	(*FB_Gripper Manual*)
		fbGripperManu( // Call Griper mouvement
				eGripperMode:=eGripperMode,
				tMouvementDuration:=tGripperTime,
				bSensorCheck:=bGripperSensor
				);
		IF fbGripperManu.bDone THEN // Gripper Done
			fbGripperManu.bStart:=FALSE;
			(*Log*)
				PRG_Log_WM.fbLogWM.M_Write_Log('MANUAL : Gripper -> DONE');
		ELSIF fbGripperManu.bError THEN // Gripper Error
			//bError:=TRUE;
			//udiErrorID:=?00+fbGripper.udiErrorID; // ?xx = ? + Error xx fbGripperManu
			fbGripperManu.bStart:=FALSE;
			(*Log*)
				PRG_Log_WM.fbLogWM.M_Write_Log('MANUAL : GripperUnclamp -> ERROR');
				PRG_Log_WM.fbLogWM.M_Write_Log(CONCAT('MANUAL : GripperUnclamp : ErrorID=',UDINT_TO_STRING(fbGripperManu.udiErrorID)));
		END_IF
			
(** CHANGING ARM **)
	(*Axis Position*)
		GV_Tool_Magazine.stArm.lrArmPosition:=LINT_TO_LREAL(LREAL_TO_LINT(GV_Axes.stAxisArm.stDriveAx8206.AxisRef.NcToPlc.ActPos*1000.0))/1000.0;
	(*Memory*)
		(*Gripper1*)
			IF GV_Tool_Magazine.stArm.aGripper[1].iAbsLocationNumberMemory<>0 AND GV_Tool_Magazine.stArm.aGripper[1].iRelLocationNumberMemory<>0 THEN
				GV_Tool_Magazine.stArm.aGripper[1].bToolPresenceMemory:=TRUE;
			ELSE
				GV_Tool_Magazine.stArm.aGripper[1].bToolPresenceMemory:=FALSE;
			END_IF
		(*Gripper2*)
			IF GV_Tool_Magazine.stArm.aGripper[2].iAbsLocationNumberMemory<>0 AND GV_Tool_Magazine.stArm.aGripper[2].iRelLocationNumberMemory<>0 THEN
				GV_Tool_Magazine.stArm.aGripper[2].bToolPresenceMemory:=TRUE;
			ELSE
				GV_Tool_Magazine.stArm.aGripper[2].bToolPresenceMemory:=FALSE;
			END_IF
	(*Positions*)
		IF GV_Tool_Magazine.stArm.lrArmPosition<=(GV_Tool_Magazine.stArm.lrArmHome+GV_Tool_Magazine.stArm.lrArmPositionTol) AND GV_Tool_Magazine.stArm.lrArmPosition>=(GV_Tool_Magazine.stArm.lrArmHome-GV_Tool_Magazine.stArm.lrArmPositionTol) THEN
			GV_Tool_Magazine.stArm.ePositionAxis:=ENUM_Position_Axis.Home;
		ELSIF GV_Tool_Magazine.stArm.lrArmPosition<=(GV_Tool_Magazine.stArm.lrArmManipulator+GV_Tool_Magazine.stArm.lrArmPositionTol) AND GV_Tool_Magazine.stArm.lrArmPosition>=(GV_Tool_Magazine.stArm.lrArmManipulator-GV_Tool_Magazine.stArm.lrArmPositionTol) THEN 
			GV_Tool_Magazine.stArm.ePositionAxis:=ENUM_Position_Axis.Work1;
		ELSIF GV_Tool_Magazine.stArm.lrArmPosition<=(GV_Tool_Magazine.stArm.lrArmCNC+GV_Tool_Magazine.stArm.lrArmPositionTol) AND GV_Tool_Magazine.stArm.lrArmPosition>=(GV_Tool_Magazine.stArm.lrArmCNC-GV_Tool_Magazine.stArm.lrArmPositionTol) THEN 
			GV_Tool_Magazine.stArm.ePositionAxis:=ENUM_Position_Axis.CNC;
		ELSE
			GV_Tool_Magazine.stArm.ePositionAxis:=ENUM_Position_Axis.Unknow;
		END_IF

	(*Evacuate*)
		//IF GV_CNC.stFanucData.stCncMagazine.biEvacuateArm AND  THEN
			
		//END_IF

(** TEACHING **)
	(* Selected Location *)
		IF GV_HMI.stMagazineTeach.iTeachLocationSelected>0 AND (GV_HMI.stMagazineTeach.iTeachLocationSelected+1)<=GV_Tool_Magazine.iMaxAbsLocation THEN
			GV_HMI.stMagazineTeach.sTeachLocationSelected:=INT_TO_STRING(GV_Tool_Magazine.aLocation[(GV_HMI.stMagazineTeach.iTeachLocationSelected+1)].iRelLocationNumber);
		END_IF
	
	(* Authorization *)
		GV_Tool_Magazine.bAuthorizationTeachLocation:=(NOT GV_Cycle.bCycleInProgress) AND GV_OpMode.eOpMode=ENUM_OpMode.MANU AND GV_Axes.bAxisAllNotMoving AND (*GV_Axes.bAxisAllOperational AND*) GV_HMI.iCurrentScreenNumber=310 AND GV_HMI.stMagazineTeach.iTeachLocationSelected>0 AND (GV_HMI.stMagazineTeach.iTeachLocationSelected+1)<=GV_Tool_Magazine.iMaxAbsLocation;
		GV_Tool_Magazine.bAuthorizationTeachRack:=(NOT GV_Cycle.bCycleInProgress) AND GV_HMI.iCurrentScreenNumber=310;
		GV_Tool_Magazine.bAuthorizationTeachAllTop:=(NOT GV_Cycle.bCycleInProgress) AND GV_HMI.iCurrentScreenNumber=310;
		GV_Tool_Magazine.bAuthorizationTeachAllBottom:=(NOT GV_Cycle.bCycleInProgress) AND GV_HMI.iCurrentScreenNumber=310;
		GV_Tool_Magazine.bAuthorizationTeachPositions:=(NOT GV_Cycle.bCycleInProgress) AND GV_HMI.iCurrentScreenNumber=311;
	
	(* Limit *)
		IF GV_HMI.stMagazineTeach.iTeachLocationSelected>0 AND (GV_HMI.stMagazineTeach.iTeachLocationSelected+1)<=GV_Tool_Magazine.iMaxAbsLocation THEN
			IF GV_Tool_Magazine.aLocation[(GV_HMI.stMagazineTeach.iTeachLocationSelected+1)].ePositionMag=ENUM_Position_Magazine.Top THEN
				GV_Tool_Magazine.lrMinXTeach:=GV_Tool_Magazine.lrMinXFirstLocationTop;
				GV_Tool_Magazine.lrMaxXTeach:=GV_Tool_Magazine.lrMaxXFirstLocationTop;
				GV_Tool_Magazine.lrMinYTeach:=GV_Tool_Magazine.lrMinYLocationTop;
				GV_Tool_Magazine.lrMaxYTeach:=GV_Tool_Magazine.lrMaxYLocationTop;
				GV_Tool_Magazine.lrMinZTeach:=GV_Tool_Magazine.lrMinZLowestRackTop;
				GV_Tool_Magazine.lrMaxZTeach:=GV_Tool_Magazine.lrMaxZLowestRackTop;
			ELSIF GV_Tool_Magazine.aLocation[(GV_HMI.stMagazineTeach.iTeachLocationSelected+1)].ePositionMag=ENUM_Position_Magazine.Bottom THEN
				GV_Tool_Magazine.lrMinXTeach:=GV_Tool_Magazine.lrMinXFirstLocationBottom;
				GV_Tool_Magazine.lrMaxXTeach:=GV_Tool_Magazine.lrMaxXFirstLocationBottom;
				GV_Tool_Magazine.lrMinYTeach:=GV_Tool_Magazine.lrMinYLocationBottom;
				GV_Tool_Magazine.lrMaxYTeach:=GV_Tool_Magazine.lrMaxYLocationBottom;
				GV_Tool_Magazine.lrMinZTeach:=GV_Tool_Magazine.lrMinZLowestRackBottom;
				GV_Tool_Magazine.lrMaxZTeach:=GV_Tool_Magazine.lrMaxZLowestRackBottom;
			ELSE
				GV_Tool_Magazine.lrMinXTeach:=9999.999;
				GV_Tool_Magazine.lrMaxXTeach:=9999.999;
				GV_Tool_Magazine.lrMinYTeach:=9999.999;
				GV_Tool_Magazine.lrMaxYTeach:=9999.999;
				GV_Tool_Magazine.lrMinZTeach:=9999.999;
				GV_Tool_Magazine.lrMaxZTeach:=9999.999;
			END_IF
		END_IF
		
	(* Teach Location *)
		IF GV_HMI.stMagazineTeach.rtTeachLocation.Q AND GV_Tool_Magazine.bAuthorizationTeachLocation AND GV_HMI.stMagazineTeach.iTeachLocationSelected>0 AND (GV_HMI.stMagazineTeach.iTeachLocationSelected+1)<=GV_Tool_Magazine.iMaxAbsLocation THEN
			GV_Tool_Magazine.aLocation[(GV_HMI.stMagazineTeach.iTeachLocationSelected+1)].lrXcoord:=LINT_TO_LREAL(LREAL_TO_LINT(GV_Axes.stAxisX.stDriveAx8206.AxisRef.NcToPlc.ActPos*1000.0))/1000.0; // Round 10e-3
			GV_Tool_Magazine.aLocation[(GV_HMI.stMagazineTeach.iTeachLocationSelected+1)].lrYcoord:=LINT_TO_LREAL(LREAL_TO_LINT(GV_Axes.stAxisY.stDriveAx8206.AxisRef.NcToPlc.ActPos*1000.0))/1000.0; // Round 10e-3
			GV_Tool_Magazine.aLocation[(GV_HMI.stMagazineTeach.iTeachLocationSelected+1)].lrZcoord:=LINT_TO_LREAL(LREAL_TO_LINT(GV_Axes.stAxisZ.stDriveAx8206.AxisRef.NcToPlc.ActPos*1000.0))/1000.0; // Round 10e-3
		END_IF

	(* Teach Rack *)
		IF GV_HMI.stMagazineTeach.iTeachLocationSelected>0 AND (GV_HMI.stMagazineTeach.iTeachLocationSelected+1)<=GV_Tool_Magazine.iMaxAbsLocation THEN
			
			IF GV_Tool_Magazine.aLocation[(GV_HMI.stMagazineTeach.iTeachLocationSelected+1)].iRelLocationNumber>1 THEN
				IF GV_Tool_Magazine.aLocation[(GV_HMI.stMagazineTeach.iTeachLocationSelected)].iRackNumber<GV_Tool_Magazine.aLocation[(GV_HMI.stMagazineTeach.iTeachLocationSelected+1)].iRackNumber THEN
					GV_HMI.stMagazineTeach.bVisuTeachRack:=TRUE;
				ELSE
					IF GV_Tool_Magazine.aLocation[(GV_HMI.stMagazineTeach.iTeachLocationSelected)].iRackNumber=GV_Tool_Magazine.aLocation[(GV_HMI.stMagazineTeach.iTeachLocationSelected+1)].iRackNumber AND GV_Tool_Magazine.aLocation[(GV_HMI.stMagazineTeach.iTeachLocationSelected)].iRelLocationNumber=0 THEN
						GV_HMI.stMagazineTeach.bVisuTeachRack:=TRUE;
					ELSE
						GV_HMI.stMagazineTeach.bVisuTeachRack:=FALSE;
					END_IF
				END_IF
			ELSE
				IF GV_Tool_Magazine.aLocation[(GV_HMI.stMagazineTeach.iTeachLocationSelected+1)].iRelLocationNumber=1 THEN
					GV_HMI.stMagazineTeach.bVisuTeachRack:=TRUE;
				ELSE
					GV_HMI.stMagazineTeach.bVisuTeachRack:=FALSE;
				END_IF
			END_IF
			
			IF GV_HMI.stMagazineTeach.rtTeachRack.Q AND GV_HMI.stMagazineTeach.bVisuTeachRack AND GV_Tool_Magazine.bAuthorizationTeachRack THEN
				IF GV_Tool_Magazine.aLocation[(GV_HMI.stMagazineTeach.iTeachLocationSelected+1)].ePositionMag=ENUM_Position_magazine.Top THEN
					iCount:=0;
					lrTeachRackZ:=0;
					FOR iTeachLoop:=(GV_HMI.stMagazineTeach.iTeachLocationSelected+1) TO GV_Tool_Magazine.iMaxAbsLocation BY 1 DO
						IF iTeachLoop=(GV_HMI.stMagazineTeach.iTeachLocationSelected+1) THEN
							lrTeachRackZ:=GV_Tool_Magazine.aLocation[(GV_HMI.stMagazineTeach.iTeachLocationSelected+1)].lrZcoord;
						END_IF
						IF GV_Tool_Magazine.aLocation[iTeachLoop].iRackNumber=GV_Tool_Magazine.aLocation[(GV_HMI.stMagazineTeach.iTeachLocationSelected+1)].iRackNumber THEN
							GV_Tool_Magazine.aLocation[iTeachLoop].lrXcoord:=GV_Tool_Magazine.aLocation[(GV_HMI.stMagazineTeach.iTeachLocationSelected+1)].lrXcoord+(GV_Tool_Magazine.lrXLocationOffsetTop*(iTeachLoop-(GV_HMI.stMagazineTeach.iTeachLocationSelected+1)));
								GV_Tool_Magazine.aLocation[iTeachLoop].lrXcoord:=LINT_TO_LREAL(LREAL_TO_LINT(GV_Tool_Magazine.aLocation[iTeachLoop].lrXcoord*1000.0))/1000.0; // Round 10e-3
							GV_Tool_Magazine.aLocation[iTeachLoop].lrYcoord:=GV_Tool_Magazine.aLocation[(GV_HMI.stMagazineTeach.iTeachLocationSelected+1)].lrYcoord+(GV_Tool_Magazine.lrYLocationOffsetTop*(iTeachLoop-(GV_HMI.stMagazineTeach.iTeachLocationSelected+1)));;
								GV_Tool_Magazine.aLocation[iTeachLoop].lrYcoord:=LINT_TO_LREAL(LREAL_TO_LINT(GV_Tool_Magazine.aLocation[iTeachLoop].lrYcoord*1000.0))/1000.0; // Round 10e-3
 							GV_Tool_Magazine.aLocation[iTeachLoop].lrZcoord:=lrTeachRackZ-(GV_Tool_Magazine.lrZRelCompensationLocationTop*iCount); // Compensation
								GV_Tool_Magazine.aLocation[iTeachLoop].lrZcoord:=LINT_TO_LREAL(LREAL_TO_LINT(GV_Tool_Magazine.aLocation[iTeachLoop].lrZcoord*1000.0))/1000.0; // Round 10e-3
							iCount:=iCount+1;
						ELSE
							EXIT;
						END_IF
					END_FOR
				ELSIF GV_Tool_Magazine.aLocation[(GV_HMI.stMagazineTeach.iTeachLocationSelected+1)].ePositionMag=ENUM_Position_magazine.Bottom THEN
					iCount:=0;
					lrTeachRackZ:=0;
					FOR iTeachLoop:=(GV_HMI.stMagazineTeach.iTeachLocationSelected+1) TO GV_Tool_Magazine.iMaxAbsLocation BY 1 DO
						IF iTeachLoop=(GV_HMI.stMagazineTeach.iTeachLocationSelected+1) THEN
							lrTeachRackZ:=GV_Tool_Magazine.aLocation[(GV_HMI.stMagazineTeach.iTeachLocationSelected+1)].lrZcoord;
						END_IF
						IF GV_Tool_Magazine.aLocation[iTeachLoop].iRackNumber=GV_Tool_Magazine.aLocation[(GV_HMI.stMagazineTeach.iTeachLocationSelected+1)].iRackNumber THEN
							GV_Tool_Magazine.aLocation[iTeachLoop].lrXcoord:=GV_Tool_Magazine.aLocation[(GV_HMI.stMagazineTeach.iTeachLocationSelected+1)].lrXcoord+(GV_Tool_Magazine.lrXLocationOffsetBottom*(iTeachLoop-(GV_HMI.stMagazineTeach.iTeachLocationSelected+1)));
								GV_Tool_Magazine.aLocation[iTeachLoop].lrXcoord:=LINT_TO_LREAL(LREAL_TO_LINT(GV_Tool_Magazine.aLocation[iTeachLoop].lrXcoord*1000.0))/1000.0; // Round 10e-3
							GV_Tool_Magazine.aLocation[iTeachLoop].lrYcoord:=GV_Tool_Magazine.aLocation[(GV_HMI.stMagazineTeach.iTeachLocationSelected+1)].lrYcoord+(GV_Tool_Magazine.lrYLocationOffsetBottom*(iTeachLoop-(GV_HMI.stMagazineTeach.iTeachLocationSelected+1)));
								GV_Tool_Magazine.aLocation[iTeachLoop].lrYcoord:=LINT_TO_LREAL(LREAL_TO_LINT(GV_Tool_Magazine.aLocation[iTeachLoop].lrYcoord*1000.0))/1000.0; // Round 10e-3
							GV_Tool_Magazine.aLocation[iTeachLoop].lrZcoord:=lrTeachRackZ-(GV_Tool_Magazine.lrZRelCompensationLocationBottom*iCount); // Compensation
								GV_Tool_Magazine.aLocation[iTeachLoop].lrZcoord:=LINT_TO_LREAL(LREAL_TO_LINT(GV_Tool_Magazine.aLocation[iTeachLoop].lrZcoord*1000.0))/1000.0; // Round 10e-3
							iCount:=iCount+1;
						ELSE
							EXIT;
						END_IF
					END_FOR
				//ELSE
					// Normally not possible to be here -> Can't select from HMI a Location with (ENUM_Position_magazine<>Top OR ENUM_Position_magazine<>Bottom)
				END_IF
			END_IF
			
		END_IF
	
	(* Teach All Top *)
// 		IF GV_HMI.stMagazineTeach.iTeachLocationSelected>0 AND (GV_HMI.stMagazineTeach.iTeachLocationSelected+1)<=GV_Tool_Magazine.iMaxAbsLocation THEN
// 			
// 			IF GV_Tool_Magazine.aLocation[(GV_HMI.stMagazineTeach.iTeachLocationSelected+1)].iRelLocationNumber=1 AND GV_Tool_Magazine.aLocation[(GV_HMI.stMagazineTeach.iTeachLocationSelected+1)].ePositionMag=ENUM_Position_magazine.Top THEN
// 				IF GV_Tool_Magazine.aLocation[(GV_HMI.stMagazineTeach.iTeachLocationSelected+1)].iRackNumber = 1eR Rack du haut THEN
// 					GV_HMI.stMagazineTeach.bVisuTeachAllTop:=TRUE;
// 				ELSE
// 					GV_HMI.stMagazineTeach.bVisuTeachAllTop:=FALSE;
// 				END_IF
// 			ELSE
// 				GV_HMI.stMagazineTeach.bVisuTeachAllTop:=FALSE;
// 			END_IF
// 	
// 			IF GV_HMI.stMagazineTeach.rtTeachAllTop.Q AND GV_HMI.stMagazineTeach.bVisuTeachAllTop AND GV_Tool_Magazine.bAuthorizationTeachAllTop THEN
// 				iCount:=0;
// 				lrTeachAllX:=0.0;
// 				lrTeachAllY:=0.0;
// 				lrTeachAllZ:=0.0;
// 				
// 				
// 				FOR iTeachLoop:=1 TO GV_Tool_Magazine.iMaxAbsLocationTop BY 1 DO
// 					
// 					// Ne pas modifier la position rel 1 car apprise, on part justement de ces valeurs pour recalculer le reste
// 					
// // 					IF iTeachLoop=(GV_HMI.stMagazineTeach.iTeachLocationSelected+1) THEN
// // 						lrTeachRackZ:=GV_Tool_Magazine.aLocation[(GV_HMI.stMagazineTeach.iTeachLocationSelected+1)].lrZcoord;
// // 					END_IF
// // 					IF GV_Tool_Magazine.aLocation[iTeachLoop].iRackNumber=GV_Tool_Magazine.aLocation[(GV_HMI.stMagazineTeach.iTeachLocationSelected+1)].iRackNumber THEN
// // 						GV_Tool_Magazine.aLocation[iTeachLoop].lrXcoord:=GV_Tool_Magazine.aLocation[(GV_HMI.stMagazineTeach.iTeachLocationSelected+1)].lrXcoord+(GV_Tool_Magazine.lrXLocationOffsetTop*(iTeachLoop-(GV_HMI.stMagazineTeach.iTeachLocationSelected+1)));
// // 							GV_Tool_Magazine.aLocation[iTeachLoop].lrXcoord:=LINT_TO_LREAL(LREAL_TO_LINT(GV_Tool_Magazine.aLocation[iTeachLoop].lrXcoord*1000.0))/1000.0; // Round 10e-3
// // 						GV_Tool_Magazine.aLocation[iTeachLoop].lrYcoord:=GV_Tool_Magazine.aLocation[(GV_HMI.stMagazineTeach.iTeachLocationSelected+1)].lrYcoord+(GV_Tool_Magazine.lrYLocationOffsetTop*(iTeachLoop-(GV_HMI.stMagazineTeach.iTeachLocationSelected+1)));;
// // 							GV_Tool_Magazine.aLocation[iTeachLoop].lrYcoord:=LINT_TO_LREAL(LREAL_TO_LINT(GV_Tool_Magazine.aLocation[iTeachLoop].lrYcoord*1000.0))/1000.0; // Round 10e-3
// //  						GV_Tool_Magazine.aLocation[iTeachLoop].lrZcoord:=lrTeachRackZ-(GV_Tool_Magazine.lrZRelCompensationLocationTop*iCount); // Compensation
// // 							GV_Tool_Magazine.aLocation[iTeachLoop].lrZcoord:=LINT_TO_LREAL(LREAL_TO_LINT(GV_Tool_Magazine.aLocation[iTeachLoop].lrZcoord*1000.0))/1000.0; // Round 10e-3
// // 						iCount:=iCount+1;
// // 					ELSE
// // 						EXIT;
// // 					END_IF
// 				END_FOR
// 				
// 				
// 				
// 			END_IF
// 	
// 		END_IF

	(* Teach All Bottom *)

END_PROGRAM

// ---- 09_Tool_Magazine/03_POUs/02_FBs/FB_Manipulator_Tunnel_5.TcPOU
FUNCTION_BLOCK FB_Manipulator_Tunnel_5
VAR_INPUT
	(** SETUP ENUM **)
		eTunnelMode : ENUM_Tunnel_Mode ; // Mode of the tunnel	

	(** SETUP TIME **)
		tTimeout : TIME ; // Max time for travel the tunnel

	(** PROCESS FLAG **)
		bInit : BOOL ; // Init the FB
	    bStart : BOOL ; // Start the Fb
END_VAR
VAR_OUTPUT
	(** PROCESS UDINT **)
		udiErrorID : UDINT ; // Fb Error ID
		
	(** PROCESS FLAG **)
		bBusy  : BOOL ; // Fb is Busy
		bDone  : BOOL ; // Fb is Done
		bError : BOOL ; // Fb in Error
END_VAR
VAR_IN_OUT
END_VAR	
VAR
	(** STRING **)
		strTextLog : STRING ; // Text to Log

	(** PROCESS INT **)
		iStep  : INT := 0 ; // Step of the Fb
		iSubStep : INT := 0 ; // SubStep of the Fb
		iPrevStep : INT := 0 ; // Previous Step of the Fb
		iPrevSubStep : INT := 0 ; // Previous Subtep of the Fb
	
	(** PROCESS FLAG + R_TRIG **)
		rtInit : R_TRIG ; // FB Init at rising edge
		rtStart : R_TRIG ; // FB Start at rising edge
		bTunnelTravelDone : BOOL ; // Tunnel travel done
		bXError : BOOL ; // Axis X Error
		bYError : BOOL ; // Axis Y Error
		bZError : BOOL ; // Axis Z Error
		bArmError : BOOL ; // Axis Arm Error
		
	(** FB **)
		tonTimeout : TON ; // TON timeout of the tunnel travel
END_VAR

//-----------------------------------------------------------------------------------------
//
//                  		FB_Manipulator_Tunnel
//
//			Management of the manipulator passage through the tunnel
//-----------------------------------------------------------------------------------------
//
//Auteur: G.GOETZ
//Création: 06.02.2026
//Dernière modification : 08.04.2026 (G.GOETZ)
//       			
//-----------------------------------------------------------------------------------------
//
//     							Liste des modifications  	
//
// 06.02.2026 (G.GOETZ) -> Création
// 08.04.2026 (G.GOETZ) -> Ajout Init + Modification du cycle
//-----------------------------------------------------------------------------------------

(** FB CALL **)
	rtInit(CLK:=bInit);
	rtStart(CLK:=bStart);
	
	tonTimeout();

(** AXIS ERRORS **)
	bXError:=(GV_Axes.stAxisX.stDriveAx8206.AxisRef.Status.Error OR GV_Axes.stAxisX.stDriveAx8206.AxisRef.Status.ErrorStop OR GV_Axes.stAxisX.stDriveAx8206.AxisRef.Status.ErrorID<>0);
	bYError:=(GV_Axes.stAxisY.stDriveAx8206.AxisRef.Status.Error OR GV_Axes.stAxisY.stDriveAx8206.AxisRef.Status.ErrorStop OR GV_Axes.stAxisY.stDriveAx8206.AxisRef.Status.ErrorID<>0);
	bZError:=(GV_Axes.stAxisZ.stDriveAx8206.AxisRef.Status.Error OR GV_Axes.stAxisZ.stDriveAx8206.AxisRef.Status.ErrorStop OR GV_Axes.stAxisZ.stDriveAx8206.AxisRef.Status.ErrorID<>0);
	bArmError:=(GV_Axes.stAxisArm.stDriveAx8206.AxisRef.Status.Error OR GV_Axes.stAxisArm.stDriveAx8206.AxisRef.Status.ErrorStop OR GV_Axes.stAxisArm.stDriveAx8206.AxisRef.Status.ErrorID<>0);

(** INIT **)
	IF (rtinit.Q OR bInit) AND (NOT bStart) THEN
		iStep:=0;
		bInit:=FALSE;
	END_IF

(** STEPS **)
    CASE iStep OF
		
        0: (* Step 0 = Idle *)
            bBusy:=FALSE;
            bDone:=FALSE;
			bError:=FALSE;
			udiErrorID:=0;
			iSubStep:=0;
			
			tonTimeout.IN:=FALSE;
			
			bTunnelTravelDone:=FALSE;
			
			(* Idle->Setup *)
				IF bStart AND (NOT bInit) THEN
					bBusy:=TRUE;
					(*Log*)
						PRG_Log_WM.fbLogWM.M_Write_Log('FB_Manipulator_Tunnel : 0_Idle->1_Setup');
					iStep:=1; // Next Step
				END_IF
				
		1: (* Step 1 = Setup *)
			(*Log*)
				(*TunnelMode*)
					CASE eTunnelMode OF
						ENUM_Tunnel_Mode.TopToBottom:		strTextLog:='TopToBottom';
						ENUM_Tunnel_Mode.BottomToTop:		strTextLog:='BottomToTop';
					END_CASE
					PRG_Log_WM.fbLogWM.M_Write_Log(CONCAT('FB_Manipulator_Tunnel : 1_Setup : Tunnel Mode = ',strTextLog));
				(*Timeout*)
					strTextLog:=TIME_TO_STRING(tTimeout);
					PRG_Log_WM.fbLogWM.M_Write_Log(CONCAT('FB_Manipulator_Tunnel : 1_Setup : Timeout = ',strTextLog));				
				PRG_Log_WM.fbLogWM.M_Write_Log('FB_Manipulator_Tunnel : 1_Setup->2_Process');
				
			tonTimeout.PT:=tTimeout;
			iStep:=2; // Next Step
			
		2: (* Step 2 = Process (Y->(XFirst)->Z->X) *) // -> (* Step 2 = Process (Y->(ZLowestRacKTop)->(XFirst)) *) + (* Step 3 = Process (Z->X) *)	
			tonTimeout.IN:=TRUE; // Start TON timeout

				CASE iSubStep OF
		
					0: (* Start Y move *)
						GV_Axes.stAxisY.lrAutoPosAbs:=GV_Tool_Magazine.stManipulator.lrYTunnel;
						GV_Axes.stAxisY.bAutoCmdAbs:=TRUE;
						(*Log*)
							PRG_Log_WM.fbLogWM.M_Write_Log('FB_Manipulator_Tunnel : 2_Process : 0 : Start Y move');
						iSubStep:=1; // Next SubStep
						
					1: (* Wait Y move done *)
					   IF GV_Axes.stAxisY.bAutoDone AND (NOT bYError) THEN
							GV_Axes.stAxisY.bAutoCmdAbs:=FALSE;
							(*Log*)
								PRG_Log_WM.fbLogWM.M_Write_Log('FB_Manipulator_Tunnel : 2_Process : 1 : Y move done');

							CASE eTunnelMode OF 
								ENUM_Tunnel_Mode.TopToBottom: // X Top
									IF GV_Tool_Magazine.stManipulator.lrXPosition<GV_Tool_Magazine.lrXFirstLocationTop THEN
										(*Log*)
											PRG_Log_WM.fbLogWM.M_Write_Log('FB_Manipulator_Tunnel : 2_Process : 1->2 : XFirstTop');
										iSubStep:=2; // Next SubStep
									ELSE
										(*Log*)
											PRG_Log_WM.fbLogWM.M_Write_Log('FB_Manipulator_Tunnel : 2_Process : 1->4 : Z');
										iSubStep:=4; // Next SubStep
									END_IF
								ENUM_Tunnel_Mode.BottomToTop: // X Bottom
									IF GV_Tool_Magazine.stManipulator.lrXPosition<GV_Tool_Magazine.lrXFirstLocationBottom THEN
										(*Log*)
											PRG_Log_WM.fbLogWM.M_Write_Log('FB_Manipulator_Tunnel : 2_Process : 1->2 : XFirstBottom');
										iSubStep:=2; // Next SubStep
									ELSE
										(*Log*)
											PRG_Log_WM.fbLogWM.M_Write_Log('FB_Manipulator_Tunnel : 2_Process : 1->4 : Z');
										iSubStep:=4; // Next SubStep
									END_IF
							END_CASE
						ELSIF bYError THEN
							bError:=TRUE;
							udiErrorID:=21; // 21 = Step 2 SubStep 1 Error Axis Y
							GV_Axes.stAxisY.bAutoCmdAbs:=FALSE;
							tonTimeout.IN:=FALSE;
							(*Log*)
								PRG_Log_WM.fbLogWM.M_Write_Log('FB_Manipulator_Tunnel : 2_Process=Error');
								PRG_Log_WM.fbLogWM.M_Write_Log(CONCAT('FB_Manipulator_Tunnel : ErrorID=',UDINT_TO_STRING(udiErrorID)));
							iSubStep:=0; // Stop SubStep
							iStep:=0; // Idle Step
						END_IF
						
					2: (* Start XFirst move *)
						CASE eTunnelMode OF 
							ENUM_Tunnel_Mode.TopToBottom: // X Top
								GV_Axes.stAxisX.lrAutoPosAbs:=GV_Tool_Magazine.lrXFirstLocationTop;
								(*Log*)
									PRG_Log_WM.fbLogWM.M_Write_Log('FB_Manipulator_Tunnel : 2_Process : 2 : Start XFirstTop move');
							ENUM_Tunnel_Mode.BottomToTop: // X Bottom
								GV_Axes.stAxisX.lrAutoPosAbs:=GV_Tool_Magazine.lrXFirstLocationBottom;
								(*Log*)
									PRG_Log_WM.fbLogWM.M_Write_Log('FB_Manipulator_Tunnel : 2_Process : 2 : Start XFirstBottom move');
						END_CASE
						GV_Axes.stAxisX.bAutoCmdAbs:=TRUE;
						iSubStep:=3; // Next SubStep

					3: (* Wait XFirst move done *)
					   IF GV_Axes.stAxisX.bAutoDone AND (NOT bXError) THEN
							GV_Axes.stAxisX.bAutoCmdAbs:=FALSE;
							(*Log*)
								PRG_Log_WM.fbLogWM.M_Write_Log('FB_Manipulator_Tunnel : 2_Process : 3 : XFirst move done');
							iSubStep:=4; // Next SubStep
						ELSIF bXError THEN
							bError:=TRUE;
							udiErrorID:=23; // 23 = Step 2 SubStep 3 Error Axis X
							GV_Axes.stAxisX.bAutoCmdAbs:=FALSE;
							tonTimeout.IN:=FALSE;
							(*Log*)
								PRG_Log_WM.fbLogWM.M_Write_Log('FB_Manipulator_Tunnel : 2_Process=Error');
								PRG_Log_WM.fbLogWM.M_Write_Log(CONCAT('FB_Manipulator_Tunnel : ErrorID=',UDINT_TO_STRING(udiErrorID)));
							iSubStep:=0; // Stop 
							iStep:=0; // Idle Step
						END_IF
						
					4: (* Start Z move *)
						CASE eTunnelMode OF 
							ENUM_Tunnel_Mode.TopToBottom: // Z bottom position
								GV_Axes.stAxisZ.lrAutoPosAbs:=GV_Tool_Magazine.stManipulator.lrZTunnelBottom;
							ENUM_Tunnel_Mode.BottomToTop: // Z top position
								GV_Axes.stAxisZ.lrAutoPosAbs:=GV_Tool_Magazine.stManipulator.lrZTunnelTop;
						END_CASE
						IF (GV_Axes.stAxisZ.lrAutoPosAbs=GV_Tool_Magazine.stManipulator.lrZTunnelBottom) OR (GV_Axes.stAxisZ.lrAutoPosAbs=GV_Tool_Magazine.stManipulator.lrZTunnelTop) THEN
							GV_Axes.stAxisZ.bAutoCmdAbs:=TRUE;
						ELSE
							GV_Axes.stAxisZ.bAutoCmdAbs:=FALSE;
						END_IF
						(*Log*)
							PRG_Log_WM.fbLogWM.M_Write_Log('FB_Manipulator_Tunnel : 2_Process : 4 : Start Z move');
						iSubStep:=5; // Next Step
		
					5: (* Wait Z move done *)
					   IF GV_Axes.stAxisZ.bAutoDone AND (NOT bZError) THEN
							GV_Axes.stAxisZ.bAutoCmdAbs:=FALSE;
							tonTimeout.IN:=FALSE;
							(*Log*)
								PRG_Log_WM.fbLogWM.M_Write_Log('FB_Manipulator_Tunnel : 2_Process : 5 : Z move done');
							iSubStep:=6; // End SubStep
						ELSIF bZError THEN
							bError:=TRUE;
							udiErrorID:=25; // 25 = Step 2 SubStep 5 Error Axis Z
							GV_Axes.stAxisZ.bAutoCmdAbs:=FALSE;
							tonTimeout.IN:=FALSE;
							(*Log*)
								PRG_Log_WM.fbLogWM.M_Write_Log('FB_Manipulator_Tunnel : 2_Process=Error');
								PRG_Log_WM.fbLogWM.M_Write_Log(CONCAT('FB_Manipulator_Tunnel : ErrorID=',UDINT_TO_STRING(udiErrorID)));
							iSubStep:=0; // Stop SubStep
							iStep:=0; // Idle Step
						END_IF
						
					6: (* Start X move *)
						GV_Axes.stAxisX.lrAutoPosAbs:=GV_Tool_Magazine.stManipulator.lrXTunnel;
						GV_Axes.stAxisX.bAutoCmdAbs:=TRUE;
						(*Log*)
							PRG_Log_WM.fbLogWM.M_Write_Log('FB_Manipulator_Tunnel : 2_Process : 6 : Start X move');
						iSubStep:=7; // Next SubStep
		
					7: (* Wait X move done *)
					   IF GV_Axes.stAxisX.bAutoDone AND (NOT bXError) THEN
							GV_Axes.stAxisX.bAutoCmdAbs:=FALSE;
							(*Log*)
								PRG_Log_WM.fbLogWM.M_Write_Log('FB_Manipulator_Tunnel : 2_Process : 7 : X move done');
							bTunnelTravelDone:=TRUE;
							iSubStep:=0; // Next SubStep
						ELSIF bXError THEN
							bError:=TRUE;
							udiErrorID:=27; // 27 = Step 2 SubStep 7 Error Axis X
							GV_Axes.stAxisX.bAutoCmdAbs:=FALSE;
							tonTimeout.IN:=FALSE;
							(*Log*)
								PRG_Log_WM.fbLogWM.M_Write_Log('FB_Manipulator_Tunnel : 2_Process=Error');
								PRG_Log_WM.fbLogWM.M_Write_Log(CONCAT('FB_Manipulator_Tunnel : ErrorID=',UDINT_TO_STRING(udiErrorID)));
							iSubStep:=0; // Stop SubStep
							iStep:=0; // Idle Step
						END_IF

					END_CASE
			
			IF bTunnelTravelDone THEN
				tonTimeout.IN:=FALSE;
				(*Log*)
					PRG_Log_WM.fbLogWM.M_Write_Log('FB_Manipulator_Tunnel : 2_Process : Done with success');
					PRG_Log_WM.fbLogWM.M_Write_Log('FB_Manipulator_Tunnel : 2_Process->0_Idle');
				iSubStep:=0; // End SubStep
				iStep:=0; // Idle Step
				bDone:=TRUE;
				bBusy:=FALSE;
			END_IF
			
			IF tonTimeout.Q AND tonTimeout.PT<>T#0S THEN
				bError:=TRUE;
				udiErrorID:=29; // 29 = Step 2 Error Timeout 9
				GV_Axes.stAxisZ.bAutoCmdAbs:=FALSE;
				GV_Axes.stAxisX.bAutoCmdAbs:=FALSE;
				GV_Axes.stAxisY.bAutoCmdAbs:=FALSE;
				tonTimeout.IN:=FALSE;
				(*Log*)
					PRG_Log_WM.fbLogWM.M_Write_Log('FB_Manipulator_Tunnel : 2_Process : Error');
					PRG_Log_WM.fbLogWM.M_Write_Log(CONCAT('FB_Manipulator_Tunnel : ErrorID = ',UDINT_TO_STRING(udiErrorID)));
				iSubStep:=0; // Stop SubStep
				iStep:=0; // Idle Step
			END_IF
			
	END_CASE

END_FUNCTION_BLOCK

// ---- 09_Tool_Magazine/03_POUs/02_FBs/FB_Manipulator_Tunnel_2.TcPOU
FUNCTION_BLOCK FB_Manipulator_Tunnel_2
VAR_INPUT
	(** SETUP ENUM **)
		eTunnelMode : ENUM_Tunnel_Mode ; // Mode of the tunnel	

	(** SETUP TIME **)
		tTimeout : TIME ; // Max time for travel the tunnel

	(** PROCESS FLAG **)
		bInit : BOOL ; // Init the FB
	    bStart : BOOL ; // Start the Fb
END_VAR
VAR_OUTPUT
	(** PROCESS UDINT **)
		udiErrorID : UDINT ; // Fb Error ID
		
	(** PROCESS FLAG **)
		bBusy  : BOOL ; // Fb is Busy
		bDone  : BOOL ; // Fb is Done
		bError : BOOL ; // Fb in Error
END_VAR
VAR_IN_OUT
END_VAR	
VAR
	(** STRING **)
		strTextLog : STRING ; // Text to Log

	(** PROCESS INT **)
		iStep  : INT := 0 ; // Step of the Fb
		iSubStep : INT := 0 ; // SubStep of the Fb
		iPrevStep : INT := 0 ; // Previous Step of the Fb
		iPrevSubStep : INT := 0 ; // Previous Subtep of the Fb
	
	(** PROCESS FLAG + R_TRIG **)
		rtInit : R_TRIG ; // FB Init at rising edge
		rtStart : R_TRIG ; // FB Start at rising edge
		bTunnelTravelDone : BOOL ; // Tunnel travel done
		bXError : BOOL ; // Axis X Error
		bYError : BOOL ; // Axis Y Error
		bZError : BOOL ; // Axis Z Error
		bArmError : BOOL ; // Axis Arm Error
		
	(** FB **)
		tonTimeout : TON ; // TON timeout of the tunnel travel
END_VAR

//-----------------------------------------------------------------------------------------
//
//                  		FB_Manipulator_Tunnel
//
//			Management of the manipulator passage through the tunnel
//-----------------------------------------------------------------------------------------
//
//Auteur: G.GOETZ
//Création: 06.02.2026
//Dernière modification : 08.04.2026 (G.GOETZ)
//       			
//-----------------------------------------------------------------------------------------
//
//     							Liste des modifications  	
//
// 06.02.2026 (G.GOETZ) -> Création
// 08.04.2026 (G.GOETZ) -> Ajout Init + Modification du cycle
//-----------------------------------------------------------------------------------------

(** FB CALL **)
	rtInit(CLK:=bInit);
	rtStart(CLK:=bStart);
	
	tonTimeout();

(** AXIS ERRORS **)
	bXError:=(GV_Axes.stAxisX.stDriveAx8206.AxisRef.Status.Error OR GV_Axes.stAxisX.stDriveAx8206.AxisRef.Status.ErrorStop OR GV_Axes.stAxisX.stDriveAx8206.AxisRef.Status.ErrorID<>0);
	bYError:=(GV_Axes.stAxisY.stDriveAx8206.AxisRef.Status.Error OR GV_Axes.stAxisY.stDriveAx8206.AxisRef.Status.ErrorStop OR GV_Axes.stAxisY.stDriveAx8206.AxisRef.Status.ErrorID<>0);
	bZError:=(GV_Axes.stAxisZ.stDriveAx8206.AxisRef.Status.Error OR GV_Axes.stAxisZ.stDriveAx8206.AxisRef.Status.ErrorStop OR GV_Axes.stAxisZ.stDriveAx8206.AxisRef.Status.ErrorID<>0);
	bArmError:=(GV_Axes.stAxisArm.stDriveAx8206.AxisRef.Status.Error OR GV_Axes.stAxisArm.stDriveAx8206.AxisRef.Status.ErrorStop OR GV_Axes.stAxisArm.stDriveAx8206.AxisRef.Status.ErrorID<>0);

(** INIT **)
	IF (rtinit.Q OR bInit) AND (NOT bStart) THEN
		iStep:=0;
		bInit:=FALSE;
	END_IF

(** STEPS **)
    CASE iStep OF
		
        0: (* Step 0 = Idle *)
            bBusy:=FALSE;
            bDone:=FALSE;
			bError:=FALSE;
			udiErrorID:=0;
			iSubStep:=0;
			
			tonTimeout.IN:=FALSE;
			
			bTunnelTravelDone:=FALSE;
			
			(* Idle->Setup *)
				IF bStart AND (NOT bInit) THEN
					bBusy:=TRUE;
					(*Log*)
						PRG_Log_WM.fbLogWM.M_Write_Log('FB_Manipulator_Tunnel : 0_Idle->1_Setup');
					iStep:=1; // Next Step
				END_IF
				
		1: (* Step 1 = Setup *)
			(*Log*)
				(*TunnelMode*)
					CASE eTunnelMode OF
						ENUM_Tunnel_Mode.TopToBottom:		strTextLog:='TopToBottom';
						ENUM_Tunnel_Mode.BottomToTop:		strTextLog:='BottomToTop';
					END_CASE
					PRG_Log_WM.fbLogWM.M_Write_Log(CONCAT('FB_Manipulator_Tunnel : 1_Setup : Tunnel Mode = ',strTextLog));
				(*Timeout*)
					strTextLog:=TIME_TO_STRING(tTimeout);
					PRG_Log_WM.fbLogWM.M_Write_Log(CONCAT('FB_Manipulator_Tunnel : 1_Setup : Timeout = ',strTextLog));				
				PRG_Log_WM.fbLogWM.M_Write_Log('FB_Manipulator_Tunnel : 1_Setup->2_Process');
				
			tonTimeout.PT:=tTimeout;
			iStep:=2; // Next Step
			
		2: (* Step 2 = Process (Y->(ZLowestRacKTop)->(XFirst)) *)
			tonTimeout.IN:=TRUE; // Start TON timeout

				CASE iSubStep OF
		
					0: (* Start Y move *)
						GV_Axes.stAxisY.lrAutoPosAbs:=GV_Tool_Magazine.stManipulator.lrYTunnel;
						GV_Axes.stAxisY.bAutoCmdAbs:=TRUE;
						(*Log*)
							PRG_Log_WM.fbLogWM.M_Write_Log('FB_Manipulator_Tunnel : 2_Process : 0 : Start Y move');
						iSubStep:=1; // Next SubStep
						
					1: (* Wait Y move done *)
					   IF GV_Axes.stAxisY.bAutoDone AND (NOT bYError) THEN
							GV_Axes.stAxisY.bAutoCmdAbs:=FALSE;
							(*Log*)
								PRG_Log_WM.fbLogWM.M_Write_Log('FB_Manipulator_Tunnel : 2_Process : 1 : Y move done');

							CASE eTunnelMode OF 
								ENUM_Tunnel_Mode.TopToBottom: // X Top
									IF GV_Tool_Magazine.stManipulator.lrZPosition<GV_Tool_Magazine.lrZLowestRackTop THEN
										(*Log*)
											PRG_Log_WM.fbLogWM.M_Write_Log('FB_Manipulator_Tunnel : 2_Process : 1->2 : ZLowestRackTop');
										iSubStep:=2; // Next SubStep
									ELSE
										IF GV_Tool_Magazine.stManipulator.lrXPosition<GV_Tool_Magazine.lrXFirstLocationTop THEN
											(*Log*)
												PRG_Log_WM.fbLogWM.M_Write_Log('FB_Manipulator_Tunnel : 2_Process : 1->4 : XFirstTop');
											iSubStep:=4; // Next SubStep
										ELSE
											(*Log*)
												PRG_Log_WM.fbLogWM.M_Write_Log('FB_Manipulator_Tunnel : 2_Process -> 3_Process');
											iSubStep:=0; // End SubStep
											iStep:=3; // Next Stpe
										END_IF
									END_IF
								ENUM_Tunnel_Mode.BottomToTop: // X Bottom
									IF GV_Tool_Magazine.stManipulator.lrXPosition<GV_Tool_Magazine.lrXFirstLocationBottom+GV_Tool_Magazine.lrXLocationOffsetBottom THEN
										(*Log*)
											PRG_Log_WM.fbLogWM.M_Write_Log('FB_Manipulator_Tunnel : 2_Process : 1->4 : XFirstBottom');
										iSubStep:=4; // Next SubStep
									ELSE
										(*Log*)
											PRG_Log_WM.fbLogWM.M_Write_Log('FB_Manipulator_Tunnel : 2_Process -> 3_Process');
											iSubStep:=0; // End SubStep
											iStep:=3; // Next Stpe
									END_IF
							END_CASE
						ELSIF bYError THEN
							bError:=TRUE;
							udiErrorID:=21; // 21 = Step 2 SubStep 1 Error Axis Y
							GV_Axes.stAxisY.bAutoCmdAbs:=FALSE;
							tonTimeout.IN:=FALSE;
							(*Log*)
								PRG_Log_WM.fbLogWM.M_Write_Log('FB_Manipulator_Tunnel : 2_Process=Error');
								PRG_Log_WM.fbLogWM.M_Write_Log(CONCAT('FB_Manipulator_Tunnel : ErrorID=',UDINT_TO_STRING(udiErrorID)));
							iSubStep:=0; // Stop SubStep
							iStep:=0; // Idle Step
						END_IF

					2: (* Start ZLowestRacckTop move *)
						GV_Axes.stAxisZ.lrAutoPosAbs:=GV_Tool_Magazine.lrZLowestRackTop;
						(*Log*)
							PRG_Log_WM.fbLogWM.M_Write_Log('FB_Manipulator_Tunnel : 2_Process : 2 : Start ZLowestRacckTop move');
						GV_Axes.stAxisZ.bAutoCmdAbs:=TRUE;
						iSubStep:=3; // Next SubStep

					3: (* Wait ZLowestRacckTop move done *)
					   IF GV_Axes.stAxisZ.bAutoDone AND (NOT bZError) THEN
							GV_Axes.stAxisZ.bAutoCmdAbs:=FALSE;
							(*Log*)
								PRG_Log_WM.fbLogWM.M_Write_Log('FB_Manipulator_Tunnel : 2_Process : 3 : ZLowestRacckTop move done');
							iSubStep:=0; // End SubStep
							iStep:=4; // Next STep
						ELSIF bZError THEN
							bError:=TRUE;
							udiErrorID:=23; // 23 = Step 2 SubStep 3 Error Axis Z
							GV_Axes.stAxisZ.bAutoCmdAbs:=FALSE;
							tonTimeout.IN:=FALSE;
							(*Log*)
								PRG_Log_WM.fbLogWM.M_Write_Log('FB_Manipulator_Tunnel : 2_Process=Error');
								PRG_Log_WM.fbLogWM.M_Write_Log(CONCAT('FB_Manipulator_Tunnel : ErrorID=',UDINT_TO_STRING(udiErrorID)));
							iSubStep:=0; // Stop 
							iStep:=0; // Idle Step
						END_IF
						
					4: (* Start XFirst move *)
						CASE eTunnelMode OF 
							ENUM_Tunnel_Mode.TopToBottom: // X Top
								GV_Axes.stAxisX.lrAutoPosAbs:=GV_Tool_Magazine.lrXFirstLocationTop;
								(*Log*)
									PRG_Log_WM.fbLogWM.M_Write_Log('FB_Manipulator_Tunnel : 2_Process : 4 : Start XFirstTop move');
							ENUM_Tunnel_Mode.BottomToTop: // X Bottom
								GV_Axes.stAxisX.lrAutoPosAbs:=GV_Tool_Magazine.lrXFirstLocationBottom+GV_Tool_Magazine.lrXLocationOffsetBottom;
								(*Log*)
									PRG_Log_WM.fbLogWM.M_Write_Log('FB_Manipulator_Tunnel : 2_Process : 4 : Start XFirstBottom move');
						END_CASE
						GV_Axes.stAxisX.bAutoCmdAbs:=TRUE;
						iSubStep:=5; // Next SubStep

					5: (* Wait XFirst move done *)
					   IF GV_Axes.stAxisX.bAutoDone AND (NOT bXError) THEN
							GV_Axes.stAxisX.bAutoCmdAbs:=FALSE;
							(*Log*)
								PRG_Log_WM.fbLogWM.M_Write_Log('FB_Manipulator_Tunnel : 2_Process : 5 : XFirst move done');
							iSubStep:=0; // End SubStep
							iStep:=3; // Next STep
						ELSIF bXError THEN
							bError:=TRUE;
							udiErrorID:=25; // 25 = Step 2 SubStep 5 Error Axis X
							GV_Axes.stAxisX.bAutoCmdAbs:=FALSE;
							tonTimeout.IN:=FALSE;
							(*Log*)
								PRG_Log_WM.fbLogWM.M_Write_Log('FB_Manipulator_Tunnel : 2_Process=Error');
								PRG_Log_WM.fbLogWM.M_Write_Log(CONCAT('FB_Manipulator_Tunnel : ErrorID=',UDINT_TO_STRING(udiErrorID)));
							iSubStep:=0; // Stop 
							iStep:=0; // Idle Step
						END_IF
						
				END_CASE
				
			IF tonTimeout.Q AND tonTimeout.PT<>T#0S THEN
				bError:=TRUE;
				udiErrorID:=29; // 29 = Step 2 Error Timeout 9
				GV_Axes.stAxisZ.bAutoCmdAbs:=FALSE;
				GV_Axes.stAxisX.bAutoCmdAbs:=FALSE;
				GV_Axes.stAxisY.bAutoCmdAbs:=FALSE;
				tonTimeout.IN:=FALSE;
				(*Log*)
					PRG_Log_WM.fbLogWM.M_Write_Log('FB_Manipulator_Tunnel : 2_Process : Error');
					PRG_Log_WM.fbLogWM.M_Write_Log(CONCAT('FB_Manipulator_Tunnel : ErrorID = ',UDINT_TO_STRING(udiErrorID)));
				iSubStep:=0; // Stop SubStep
				iStep:=0; // Idle Step
			END_IF
			
		3: (* Step 3 = Process (Z->X) *)	
				CASE iSubStep OF

					0: (* Start Z move *)
						CASE eTunnelMode OF 
							ENUM_Tunnel_Mode.TopToBottom: // Z bottom position
								GV_Axes.stAxisZ.lrAutoPosAbs:=GV_Tool_Magazine.stManipulator.lrZTunnelBottom;
							ENUM_Tunnel_Mode.BottomToTop: // Z top position
								GV_Axes.stAxisZ.lrAutoPosAbs:=GV_Tool_Magazine.stManipulator.lrZTunnelTop;
						END_CASE
						IF (GV_Axes.stAxisZ.lrAutoPosAbs=GV_Tool_Magazine.stManipulator.lrZTunnelBottom) OR (GV_Axes.stAxisZ.lrAutoPosAbs=GV_Tool_Magazine.stManipulator.lrZTunnelTop) THEN
							GV_Axes.stAxisZ.bAutoCmdAbs:=TRUE;
						ELSE
							GV_Axes.stAxisZ.bAutoCmdAbs:=FALSE;
						END_IF
						(*Log*)
							PRG_Log_WM.fbLogWM.M_Write_Log('FB_Manipulator_Tunnel : 3_Process : 0 : Start Z move');
						iSubStep:=1; // Next Step
		
					1: (* Wait Z move done *)
					   IF GV_Axes.stAxisZ.bAutoDone AND (NOT bZError) THEN
							GV_Axes.stAxisZ.bAutoCmdAbs:=FALSE;
							tonTimeout.IN:=FALSE;
							(*Log*)
								PRG_Log_WM.fbLogWM.M_Write_Log('FB_Manipulator_Tunnel : 2_Process : 1 : Z move done');
							iSubStep:=2; // End SubStep
						ELSIF bZError THEN
							bError:=TRUE;
							udiErrorID:=31; // 31 = Step 3 SubStep 1 Error Axis Z
							GV_Axes.stAxisZ.bAutoCmdAbs:=FALSE;
							tonTimeout.IN:=FALSE;
							(*Log*)
								PRG_Log_WM.fbLogWM.M_Write_Log('FB_Manipulator_Tunnel : 3_Process=Error');
								PRG_Log_WM.fbLogWM.M_Write_Log(CONCAT('FB_Manipulator_Tunnel : ErrorID=',UDINT_TO_STRING(udiErrorID)));
							iSubStep:=0; // Stop SubStep
							iStep:=0; // Idle Step
						END_IF
						
					2: (* Start X move *)
						GV_Axes.stAxisX.lrAutoPosAbs:=GV_Tool_Magazine.stManipulator.lrXTunnel;
						GV_Axes.stAxisX.bAutoCmdAbs:=TRUE;
						(*Log*)
							PRG_Log_WM.fbLogWM.M_Write_Log('FB_Manipulator_Tunnel : 3_Process : 2 : Start X move');
						iSubStep:=7; // Next SubStep
		
					3: (* Wait X move done *)
					   IF GV_Axes.stAxisX.bAutoDone AND (NOT bXError) THEN
							GV_Axes.stAxisX.bAutoCmdAbs:=FALSE;
							(*Log*)
								PRG_Log_WM.fbLogWM.M_Write_Log('FB_Manipulator_Tunnel : 3_Process : 3 : X move done');
							bTunnelTravelDone:=TRUE;
							iSubStep:=0; // Next SubStep
						ELSIF bXError THEN
							bError:=TRUE;
							udiErrorID:=33; // 33 = Step 3 SubStep 3 Error Axis X
							GV_Axes.stAxisX.bAutoCmdAbs:=FALSE;
							tonTimeout.IN:=FALSE;
							(*Log*)
								PRG_Log_WM.fbLogWM.M_Write_Log('FB_Manipulator_Tunnel : 3_Process=Error');
								PRG_Log_WM.fbLogWM.M_Write_Log(CONCAT('FB_Manipulator_Tunnel : ErrorID=',UDINT_TO_STRING(udiErrorID)));
							iSubStep:=0; // Stop SubStep
							iStep:=0; // Idle Step
						END_IF

					END_CASE
			
			IF bTunnelTravelDone THEN
				tonTimeout.IN:=FALSE;
				(*Log*)
					PRG_Log_WM.fbLogWM.M_Write_Log('FB_Manipulator_Tunnel : 2_Process : Done with success');
					PRG_Log_WM.fbLogWM.M_Write_Log('FB_Manipulator_Tunnel : 2_Process->0_Idle');
				iSubStep:=0; // End SubStep
				iStep:=0; // Idle Step
				bDone:=TRUE;
				bBusy:=FALSE;
			END_IF
			
			IF tonTimeout.Q AND tonTimeout.PT<>T#0S THEN
				bError:=TRUE;
				udiErrorID:=39; // 39 = Step 3 Error Timeout 9
				GV_Axes.stAxisZ.bAutoCmdAbs:=FALSE;
				GV_Axes.stAxisX.bAutoCmdAbs:=FALSE;
				GV_Axes.stAxisY.bAutoCmdAbs:=FALSE;
				tonTimeout.IN:=FALSE;
				(*Log*)
					PRG_Log_WM.fbLogWM.M_Write_Log('FB_Manipulator_Tunnel : 3_Process : Error');
					PRG_Log_WM.fbLogWM.M_Write_Log(CONCAT('FB_Manipulator_Tunnel : ErrorID = ',UDINT_TO_STRING(udiErrorID)));
				iSubStep:=0; // Stop SubStep
				iStep:=0; // Idle Step
			END_IF
			
	END_CASE

END_FUNCTION_BLOCK

// ---- 10_Axes/03_POUs/01_PRGs/PRG_Handwheel.TcPOU
PROGRAM PRG_Handwheel
VAR
	(** INT **)
		iHandwheelLoop : INT := 0 ; // INT use in a FOR Loop
	
	(** FB **)
		//FbHandwheel : FB_Handwheel ;
		FbHandwheel : FB_Handwheel_2 ;
END_VAR

//-----------------------------------------------------------------------------------------
//
//                  				PRG_Handwheel
//
//				Gestion de la manivelle déportée pour mouvement des Axes     			
//-----------------------------------------------------------------------------------------
//
//Auteur: G.GOETZ
//Création: 19.01.2026
//Dernière modification : 19.01.2026 (G.GOETZ)
//       			
//-----------------------------------------------------------------------------------------
//
//     							Liste des modifications  	
//
// 19.01.2026 (G.GOETZ) -> Création	
//-----------------------------------------------------------------------------------------

(** TOOL MAGAZINE HANDWHEEL **)
	GV_Handwheel.aId[1].bPresence:=TRUE;
	(* Enable *)
		IF GV_HMI.rtHandwheelEnable.Q THEN
			IF (NOT GV_Handwheel.aId[1].bEnable) THEN
				GV_Handwheel.aId[1].bEnable:=TRUE;
			ELSE
				GV_Handwheel.aId[1].bEnable:=FALSE;
			END_IF
		END_IF
	(* Axis selector *)
		GV_Handwheel.aId[1].bAxisSelectorB0:=GV_IO.diHandwheelAxisSelectorB0;
		GV_Handwheel.aId[1].bAxisSelectorB1:=GV_IO.diHandwheelAxisSelectorB1;
		GV_Handwheel.aId[1].bAxisSelectorB2:=GV_IO.diHandwheelAxisSelectorB2;
	(* Incremental selector *)
		GV_Handwheel.aId[1].bIncrSelectorB0:=GV_IO.diHandwheelIncrSelectorB0;
		GV_Handwheel.aId[1].bIncrSelectorB1:=GV_IO.diHandwheelIncrSelectorB1;
		GV_Handwheel.aId[1].bIncrSelectorB2:=GV_IO.diHandwheelIncrSelectorB2;
	(* Track *)
		GV_Handwheel.aId[1].bTrackA:=GV_IO.diHandwheelTrackA;
		GV_Handwheel.aId[1].bTrackB:=GV_IO.diHandwheelTrackB;
	(* Counter *)
		GV_Handwheel.aId[1].udiCounterValue:=GV_IO.udiHandwheelCounterValue;
		GV_IO.udoHandwheelCounterValue:=GV_Handwheel.aId[1].udiCounterValueSet;
		GV_Handwheel.aId[1].bCounterUnderflow:=GV_IO.biHandwheelCounterUnderflow;
		GV_Handwheel.aId[1].bCounterOverflow:=GV_IO.biHandwheelCounterOverflow;
		GV_Handwheel.aId[1].bSoftwareGateValid:=GV_IO.biSoftwareGateValid;
		GV_Handwheel.aId[1].bSetCounterDone:=GV_IO.biHandwheelSetCounterDone;
		GV_IO.boHandwheelSetCounter:=GV_Handwheel.aId[1].bSetCounter;
		GV_IO.boSoftwareGateSet:=GV_Handwheel.aId[1].bSoftwareGateSet;
	(* Button *)
		GV_Handwheel.aId[1].bButtonPlus:=GV_IO.diHandwheelButtonPlus;
		GV_Handwheel.aId[1].bButtonMinus:=GV_IO.diHandwheelButtonMinus;
		GV_Handwheel.aId[1].bButtonFast:=GV_IO.diHandwheelButtonFast;
	(* Power *)
		IF GV_Handwheel.aId[1].bPower THEN
			GV_IO.aoHandwheelPower:=GV_Handwheel.iPowerValue;
		ELSE
			GV_IO.aoHandwheelPower:=0;
		END_IF
		
(** FB_Handwheel **)
	FOR iHandwheelLoop:=1 TO GV_Handwheel.iMaxHandwheels BY 1 DO
		FbHandwheel(iHandwheelNumber:=iHandwheelLoop,StHandwheel:=GV_Handwheel.aId[iHandwheelLoop]); // Handwheel function block
	END_FOR

END_PROGRAM

// ---- 10_Axes/03_POUs/02_FBs/FB_Handwheel_2.TcPOU
FUNCTION_BLOCK FB_Handwheel_2
VAR_INPUT
	(** INT **)
		iHandwheelNumber : INT ; // Number of the handwheel
END_VAR
VAR_OUTPUT
END_VAR
VAR_IN_OUT
	(** ST **)
		stHandwheel : ST_Handwheel ;
END_VAR
VAR
	(** LREAL **)
		lrJogUnitValue : LREAL ; // Unit value for the jog
		lrJogMaxSpeed : LREAL ; // Max Speed for te Jog (in function of the Axis) (mm/s)
		lrJogMaxIncrCycle : LREAL ; // Max Incrément per PLC cycle for Jog
	
	(** DINT **)
		diCounterValueMemory : DINT ; // Memory Value of the Counter
		diDeltaPulses : DINT ; // Delta of the pulses
		diJogMaxPulseCycle : DINT ; // Max Pulse by PLC Cycle
	
	(** FLAG **)
		bChange : BOOL ;
		bJogRequest : BOOL ; // Request for Jog	
		bJogRequestMemory : BOOL ; // Memory Request for Jog	
	
	(** FB **)
		TonPowerON : TON ; // Power timer
		TonPowerOFF : TON ; // Power timer
		TonInactivity : TON ; // Inactivity timer
END_VAR

//-----------------------------------------------------------------------------------------
//
//                  				FB_Handwheel_2
//
//							Gestion manivelle(s) déportée(s)   			
//-----------------------------------------------------------------------------------------
//
//Auteur: G.GOETZ
//Création: 30.02.2026
//Dernière modification : 30.02.2026 (G.GOETZ)
//       			
//-----------------------------------------------------------------------------------------
//
//     							Liste des modifications  	
//
// 19.01.2026 (G.GOETZ) -> Création		
//-----------------------------------------------------------------------------------------

IF stHandwheel.bPresence AND stHandwheel.bEnable THEN
		
	(** EVENTS **)
	
		
	(** ALARMS **)
		
		
	(** MESSAGES **)
	//Manivelle active
	
	(** SELECTOR **) // GRAY code
		(* Axis X/Y/Z/Arm*)
			IF (NOT stHandwheel.bAxisSelectorB0) AND (NOT stHandwheel.bAxisSelectorB1) AND (NOT stHandwheel.bAxisSelectorB2) THEN // 0-0-0
				stHandwheel.eAxisSelect:=ENUM_Axis_Select.X;	
				lrJogMaxSpeed:=GV_Axes.lrJogMaxSpeedAxisX;
			ELSIF stHandwheel.bAxisSelectorB0 AND (NOT stHandwheel.bAxisSelectorB1) AND (NOT stHandwheel.bAxisSelectorB2) THEN // 1-0-0
				stHandwheel.eAxisSelect:=ENUM_Axis_Select.Y;	
				lrJogMaxSpeed:=GV_Axes.lrJogMaxSpeedAxisY;
			ELSIF stHandwheel.bAxisSelectorB0 AND stHandwheel.bAxisSelectorB1 AND (NOT stHandwheel.bAxisSelectorB2) THEN // 1-1-0
				stHandwheel.eAxisSelect:=ENUM_Axis_Select.Z;	
				lrJogMaxSpeed:=GV_Axes.lrJogMaxSpeedAxisZ;
			ELSIF (NOT stHandwheel.bAxisSelectorB0) AND stHandwheel.bAxisSelectorB1 AND (NOT stHandwheel.bAxisSelectorB2) THEN // 0-1-0
				stHandwheel.eAxisSelect:=ENUM_Axis_Select.Arm;	
				lrJogMaxSpeed:=GV_Axes.lrJogMaxSpeedAxisArm;
			ELSE
				stHandwheel.eAxisSelect:=ENUM_Axis_Select.None;
				lrJogMaxSpeed:=0.0;
			END_IF
		(* Incremental x0/x1/x10/x100/x1000*)
			IF (NOT stHandwheel.bIncrSelectorB0) AND (NOT stHandwheel.bIncrSelectorB1) AND (NOT stHandwheel.bIncrSelectorB2) THEN // 0-0-0
				stHandwheel.eIncrSelect:=ENUM_Handwheel_Incr_Select.x0;
				//stHandwheel.lrJogVel:=0.0;
				lrJogUnitValue:=0.0;
			ELSIF stHandwheel.bIncrSelectorB0 AND (NOT stHandwheel.bIncrSelectorB1) AND (NOT stHandwheel.bIncrSelectorB2) THEN // 1-0-0
				stHandwheel.eIncrSelect:=ENUM_Handwheel_Incr_Select.x1;
				//stHandwheel.lrJogVel:=(lrJogMaxSpeed/1000);
				lrJogUnitValue:=GV_Handwheel.lrUnitIncrx1;
			ELSIF stHandwheel.bIncrSelectorB0 AND stHandwheel.bIncrSelectorB1 AND (NOT stHandwheel.bIncrSelectorB2) THEN // 1-1-0
				stHandwheel.eIncrSelect:=ENUM_Handwheel_Incr_Select.x10;
				//stHandwheel.lrJogVel:=(lrJogMaxSpeed/100);
				lrJogUnitValue:=GV_Handwheel.lrUnitIncrx10;
			ELSIF (NOT stHandwheel.bIncrSelectorB0) AND stHandwheel.bIncrSelectorB1 AND (NOT stHandwheel.bIncrSelectorB2) THEN // 0-1-0
				stHandwheel.eIncrSelect:=ENUM_Handwheel_Incr_Select.x100;
				//stHandwheel.lrJogVel:=(lrJogMaxSpeed/10);
				lrJogUnitValue:=GV_Handwheel.lrUnitIncrx100;
			ELSIF (NOT stHandwheel.bIncrSelectorB0) AND stHandwheel.bIncrSelectorB1 AND stHandwheel.bIncrSelectorB2 THEN // 0-1-1
				stHandwheel.eIncrSelect:=ENUM_Handwheel_Incr_Select.x1000;
				//stHandwheel.lrJogVel:=(lrJogMaxSpeed/1);
				lrJogUnitValue:=GV_Handwheel.lrUnitIncrx1000;
			ELSE
				stHandwheel.eIncrSelect:=ENUM_Handwheel_Incr_Select.Unknow;
				//stHandwheel.lrJogVel:=0.0;
				lrJogUnitValue:=0.0;
			END_IF			

	(** POWER **)
		(* Inactivity on the handwheel *)
// 			IF stHandwheel.bButtonPlus OR stHandwheel.bButtonMinus OR stHandwheel.bButtonFast 
// 			OR (stHandwheel.eAxisSelect<>stHandwheel.eAxisSelectMemory) OR (stHandwheel.eIncrSelect<>stHandwheel.eIncrSelectMemory)
// 			OR diDeltaPulses<>0 THEN
// 				stHandwheel.bActivity:=TRUE;
// 			ELSE
// 				stHandwheel.bActivity:=FALSE;
// 			END_IF
// 			TonInactivity(IN:=(NOT stHandwheel.bActivity),PT:=GV_Handwheel.tInactivityTime);
		(* ON/OFF *)
// 			IF (NOT stHandwheel.bButtonPlus) AND (NOT stHandwheel.bButtonMinus) THEN
// 				bChange:=FALSE;
// 			END_IF
// 			TonPowerON(IN:=(stHandwheel.bButtonPlus AND stHandwheel.bButtonMinus AND (NOT stHandwheel.bPower)),PT:=GV_Handwheel.tPowerTime);
// 			TonPowerOFF(IN:=(stHandwheel.bButtonPlus AND stHandwheel.bButtonMinus AND stHandwheel.bPower),PT:=GV_Handwheel.tPowerTime);
// 			IF TonPowerON.Q AND (NOT bChange) AND (NOT GV_General.bEmergencyStop) THEN
// 				stHandwheel.bPower:=TRUE;
// 				bChange:=TRUE;
// 			END_IF
// 			IF (TonPowerOFF.Q AND (NOT bChange))THEN
// 				stHandwheel.bPower:=FALSE;
// 				bChange:=TRUE;
// 			END_IF
// 			IF TonInactivity.Q OR GV_General.bEmergencyStop THEN
// 				stHandwheel.bPower:=FALSE;
// 			END_IF	
			stHandwheel.bPower:=(stHandwheel.bEnable AND GV_General.bSafety);


	(** CONTER -> PULSE **)
		(* Max Pulse *) 
			diJogMaxPulseCycle:=MAX(1,REAL_TO_DINT(200*MAX(PRG_MAIN.lrLastExecTime_s,0.005))); // 100 pulses/tr -> 2tr/s by the human = 200pulses/s -> Task speed
		(* Ask *)
			IF stHandwheel.bSoftwareGateValid AND stHandwheel.bPower THEN // Counter is allowed
				diDeltaPulses:=(UDINT_TO_DINT(stHandwheel.udiCounterValue)-diCounterValueMemory); // Delta pulses
				diCounterValueMemory:=UDINT_TO_DINT(stHandwheel.udiCounterValue); // Memory
			ELSE
				diDeltaPulses:=0;
				diCounterValueMemory:=UDINT_TO_DINT(stHandwheel.udiCounterValue);
			END_IF
		(* Limit Pulse *)
			IF ABS(diDeltaPulses)>diJogMaxPulseCycle THEN
				diDeltaPulses:=0;
			END_IF	
	
	(** JOG **)
		(* Max Incr *) 
			//lrJogMaxIncrCycle:=MIN(lrJogMaxSpeed*PRG_MAIN.lrLastExecTime_s,lrJogUnitValue*DINT_TO_REAL(diJogMaxPulseCycle)); // Max Speed (mm/s) * Task time (s)
			lrJogMaxIncrCycle:=lrJogUnitValue*DINT_TO_REAL(diJogMaxPulseCycle);
		(* Direction *)
			IF diDeltaPulses>0 OR stHandwheel.bButtonPlus AND (NOT stHandwheel.bButtonMinus) THEN
				stHandwheel.eJogDirection:=ENUM_Jog_Direction.Plus;
			ELSIF diDeltaPulses<0 OR (NOT stHandwheel.bButtonPlus) AND stHandwheel.bButtonMinus THEN
				stHandwheel.eJogDirection:=ENUM_Jog_Direction.Minus;
			ELSE
				stHandwheel.eJogDirection:=ENUM_Jog_Direction.None;			
			END_IF
		(* Incremental Request *)
			(*Ask*)
				stHandwheel.lrJogIncrRequest:=0.0;
				IF stHandwheel.bPower AND stHandwheel.eAxisSelect<>ENUM_Axis_Select.None AND stHandwheel.eIncrSelect<>ENUM_Handwheel_Incr_Select.Unknow AND stHandwheel.eJogDirection<>ENUM_Jog_Direction.None THEN
					IF diDeltaPulses<>0 THEN
						stHandwheel.lrJogIncrRequest:=DINT_TO_REAL(diDeltaPulses)*lrJogUnitValue; // +/- X Pulse with the handwheel
						stHandwheel.eJogMode:=ENUM_Jog_Mode.Inching;
					ELSIF stHandwheel.bButtonPlus AND (NOT stHandwheel.bButtonMinus) THEN
						stHandwheel.lrJogIncrRequest:=lrJogUnitValue; // + 1 Pulse with the button (decide withe Jog direction, not here)
						stHandwheel.eJogMode:=ENUM_Jog_Mode.Inching;
						//stHandwheel.eJogMode:=ENUM_Jog_Mode.Continous;
					ELSIF (NOT stHandwheel.bButtonPlus) AND stHandwheel.bButtonMinus THEN
						stHandwheel.lrJogIncrRequest:=lrJogUnitValue; // - 1 Pulse with the button (decide withe Jog direction, not here)
						stHandwheel.eJogMode:=ENUM_Jog_Mode.Inching;
						//stHandwheel.eJogMode:=ENUM_Jog_Mode.Continous;
					ELSE
						stHandwheel.eJogMode:=ENUM_Jog_Mode.None;
					END_IF		
				ELSE
						stHandwheel.eJogMode:=ENUM_Jog_Mode.None;
				END_IF		
			(*Limit Incr*)
				IF stHandwheel.lrJogIncrRequest>lrJogMaxIncrCycle THEN
					stHandwheel.lrJogIncrRequest:=lrJogMaxIncrCycle;
				END_IF
				IF stHandwheel.lrJogIncrRequest<(-lrJogMaxIncrCycle) THEN
					stHandwheel.lrJogIncrRequest:=(-lrJogMaxIncrCycle);
				END_IF
		(* Request *)
			IF stHandwheel.bPower AND stHandwheel.eAxisSelect<>ENUM_Axis_Select.None AND stHandwheel.eIncrSelect<>ENUM_Handwheel_Incr_Select.Unknow AND stHandwheel.eJogDirection<>ENUM_Jog_Direction.None AND stHandwheel.eJogMode<>ENUM_Jog_Mode.None AND stHandwheel.lrJogIncrRequest<>0 THEN
				bJogRequest:=TRUE;
			ELSE
				bJogRequest:=FALSE;
			END_IF
			(*Rising Edge*)
				stHandwheel.bJogRequestRisingEdge:=(bJogRequest AND (NOT bJogRequestMemory));
				bJogRequestMemory:=bJogRequest;

	(** MEMORY **) // To compare and set the inactivity
		(* Axis Selector *)
			IF stHandwheel.eAxisSelect<>stHandwheel.eAxisSelectMemory THEN
				stHandwheel.eAxisSelectMemory:=stHandwheel.eAxisSelect;
			END_IF
		(* Incremental Selector *)
			IF stHandwheel.eIncrSelect<>stHandwheel.eIncrSelectMemory THEN
				stHandwheel.eIncrSelectMemory:=stHandwheel.eIncrSelect;
			END_IF

ELSE
	(** POWER **)
		(* ON/OFF *)
			stHandwheel.bPower:=FALSE;
END_IF

END_FUNCTION_BLOCK

// ---- 10_Axes/03_POUs/01_PRGs/PRG_Axis.TcPOU
PROGRAM PRG_Axis
VAR
	(** FLAG **)
		bAxisXWrite1 : BOOL ;
			rtAxisXWrite1 : R_TRIG ;
		bAxisXWrite2 : BOOL ;
			rtAxisXWrite2 : R_TRIG ;
		bAxisXWrite3 : BOOL ;
			rtAxisXWrite3 : R_TRIG ;
		bAxisXWrite4 : BOOL ;
			rtAxisXWrite4 : R_TRIG ;
		bAxisXWriteMax : BOOL ;
		bAxisXWriteMin : BOOL ;

		bAxisYWrite1 : BOOL ;
			rtAxisYWrite1 : R_TRIG ;
		bAxisYWrite2 : BOOL ;
			rtAxisYWrite2 : R_TRIG ;
		bAxisYWrite3 : BOOL ;
			rtAxisYWrite3 : R_TRIG ;
		bAxisYWrite4 : BOOL ;
			rtAxisYWrite4 : R_TRIG ;
		bAxisYWriteMax : BOOL ;
		bAxisYWriteMin : BOOL ;

		bAxisZWrite1 : BOOL ;
			rtAxisZWrite1 : R_TRIG ;
		bAxisZWrite2 : BOOL ;
			rtAxisZWrite2 : R_TRIG ;
		bAxisZWrite3 : BOOL ;
			rtAxisZWrite3 : R_TRIG ;
		bAxisZWrite4 : BOOL ;
			rtAxisZWrite4 : R_TRIG ;
		bAxisZWriteMax : BOOL ;
		bAxisZWriteMin : BOOL ;

		bAxisArmWrite1 : BOOL ;
			rtAxisArmWrite1 : R_TRIG ;
		bAxisArmWrite2 : BOOL ;
			rtAxisArmWrite2 : R_TRIG ;
		bAxisArmWrite3 : BOOL ;
			rtAxisArmWrite3 : R_TRIG ;
		bAxisArmWrite4 : BOOL ;
			rtAxisArmWrite4 : R_TRIG ;
		bAxisArmWriteMax : BOOL ;
		bAxisArmWriteMin : BOOL ;

	(** FB **)
		fbAxisX : FB_Axis ; // FB for the Axis X
		fbAxisY : FB_Axis ; // FB for the Axis Y
		fbAxisZ : FB_Axis ; // FB for the Axis Z
		fbAxisArm : FB_Axis ; // FB for the Axis Changing Arm
		fbEventGroupAssignement : FB_Event_Group_Number_Assignement ;
		
		tonZBrake : TON ;
END_VAR

//-----------------------------------------------------------------------------------------
//
//                  				PRG_Axis
//
//								Gestion des Axes   			
//-----------------------------------------------------------------------------------------
//
//Auteur: G.GOETZ
//Création: 29.01.2026
//Dernière modification : 29.01.2026 (G.GOETZ)
//       			
//-----------------------------------------------------------------------------------------
//
//     							Liste des modifications  	
//
// 29.01.2026 (G.GOETZ) -> Création		
//-----------------------------------------------------------------------------------------

(** REQUEST HMI **)
	(* Axis X *)
		IF GV_HMI.stAxes.rtButtonChoiceAxisX.Q THEN
			GV_Axes.eJogAxisRequest:=ENUM_Axis_Select.X;
		END_IF
	(* Axis Y *)
		IF GV_HMI.stAxes.rtButtonChoiceAxisY.Q THEN
			GV_Axes.eJogAxisRequest:=ENUM_Axis_Select.Y;
		END_IF
	(* Axis Z *)
		IF GV_HMI.stAxes.rtButtonChoiceAxisZ.Q THEN
			GV_Axes.eJogAxisRequest:=ENUM_Axis_Select.Z;
		END_IF
	(* Axis Arm *)
		IF GV_HMI.stAxes.rtButtonChoiceAxisArm.Q THEN
			GV_Axes.eJogAxisRequest:=ENUM_Axis_Select.Arm;
		END_IF
	(* None *)
		CASE GV_Axes.eJogAxisSelect OF
			
			ENUM_Axis_Select.X :
				IF GV_HMI.stAxes.rtButtonChoiceAxisX.Q THEN
					GV_Axes.eJogAxisRequest:=ENUM_Axis_Select.None;
				END_IF

			ENUM_Axis_Select.Y :
				IF GV_HMI.stAxes.rtButtonChoiceAxisY.Q THEN
					GV_Axes.eJogAxisRequest:=ENUM_Axis_Select.None;
				END_IF
				
			ENUM_Axis_Select.Z :
				IF GV_HMI.stAxes.rtButtonChoiceAxisZ.Q THEN
					GV_Axes.eJogAxisRequest:=ENUM_Axis_Select.None;
				END_IF
				
			ENUM_Axis_Select.Arm :
				IF GV_HMI.stAxes.rtButtonChoiceAxisArm.Q THEN
					GV_Axes.eJogAxisRequest:=ENUM_Axis_Select.None;
				END_IF

		END_CASE
		
	(* Referencing X *)
		IF GV_HMI.stAxes.rtButtonChoiceReferencingX.Q THEN
			GV_Axes.eRefAxisRequest:=ENUM_Axis_Select.X;
		END_IF
	(* Referencing Y *)
		IF GV_HMI.stAxes.rtButtonChoiceReferencingY.Q THEN
			GV_Axes.eRefAxisRequest:=ENUM_Axis_Select.Y;
		END_IF
	(* Referencing Z *)
		IF GV_HMI.stAxes.rtButtonChoiceReferencingZ.Q THEN
			GV_Axes.eRefAxisRequest:=ENUM_Axis_Select.Z;
		END_IF
	(* Referencing Arm *)
		IF GV_HMI.stAxes.rtButtonChoiceReferencingArm.Q THEN
			GV_Axes.eRefAxisRequest:=ENUM_Axis_Select.Arm;
		END_IF
	(* None *)
		CASE GV_Axes.eRefAxisSelect OF
			
			ENUM_Axis_Select.X :
				IF GV_HMI.stAxes.rtButtonChoiceReferencingX.Q THEN
					GV_Axes.eRefAxisRequest:=ENUM_Axis_Select.None;
				END_IF

			ENUM_Axis_Select.Y :
				IF GV_HMI.stAxes.rtButtonChoiceReferencingY.Q THEN
					GV_Axes.eRefAxisRequest:=ENUM_Axis_Select.None;
				END_IF
				
			ENUM_Axis_Select.Z :
				IF GV_HMI.stAxes.rtButtonChoiceReferencingZ.Q THEN
					GV_Axes.eRefAxisRequest:=ENUM_Axis_Select.None;
				END_IF
				
			ENUM_Axis_Select.Arm :
				IF GV_HMI.stAxes.rtButtonChoiceReferencingArm.Q THEN
					GV_Axes.eRefAxisRequest:=ENUM_Axis_Select.None;
				END_IF

		END_CASE
		
(** AUTHORIZATION SELECT HMI **)
	(* Axis X *)
		GV_Axes.bAxisXAllowed:=GV_General.bSafety AND GV_General.bPower AND GV_Axes.stAxisX.stDriveAx8206.AxisRef.Status.Operational AND GV_Axes.stAxisX.stDriveAx8206.AxisRef.Status.NotMoving;
	(* Axis Y *)
		GV_Axes.bAxisYAllowed:=GV_General.bSafety AND GV_General.bPower AND GV_Axes.stAxisY.stDriveAx8206.AxisRef.Status.Operational AND GV_Axes.stAxisY.stDriveAx8206.AxisRef.Status.NotMoving;
	(* Axis Z *)
		GV_Axes.bAxisZAllowed:=GV_General.bSafety AND GV_General.bPower AND GV_Axes.stAxisZ.stDriveAx8206.AxisRef.Status.Operational AND GV_Axes.stAxisZ.stDriveAx8206.AxisRef.Status.NotMoving;
	(* Axis Arm *)
		GV_Axes.bAxisArmAllowed:=GV_General.bSafety AND GV_General.bPower AND GV_Axes.stAxisArm.stDriveAx8206.AxisRef.Status.Operational AND GV_Axes.stAxisArm.stDriveAx8206.AxisRef.Status.NotMoving;

	(* Referencing X *)
		GV_Axes.bReferencingXAllowed:=GV_General.bSafety AND GV_General.bPower AND GV_Axes.stAxisX.stDriveAx8206.AxisRef.Status.Operational AND GV_Axes.stAxisX.stDriveAx8206.AxisRef.Status.NotMoving;
	(* Referencing Y *)
		GV_Axes.bReferencingYAllowed:=GV_General.bSafety AND GV_General.bPower AND GV_Axes.stAxisY.stDriveAx8206.AxisRef.Status.Operational AND GV_Axes.stAxisY.stDriveAx8206.AxisRef.Status.NotMoving;
	(* Referencing Z *)
		GV_Axes.bReferencingZAllowed:=GV_General.bSafety AND GV_General.bPower AND GV_Axes.stAxisZ.stDriveAx8206.AxisRef.Status.Operational AND GV_Axes.stAxisZ.stDriveAx8206.AxisRef.Status.NotMoving;
	(* Referencing Arm *)
		GV_Axes.bReferencingArmAllowed:=GV_General.bSafety AND GV_General.bPower AND GV_Axes.stAxisArm.stDriveAx8206.AxisRef.Status.Operational AND GV_Axes.stAxisArm.stDriveAx8206.AxisRef.Status.NotMoving;
		
(** AXIS SELECT HMI **)
	(*Transition*)
		IF GV_Axes.eJogAxisRequest<>GV_Axes.eJogAxisSelect THEN 
			CASE GV_Axes.eJogAxisRequest OF
				
				ENUM_Axis_Select.None:
					GV_Axes.eJogAxisSelect:=ENUM_Axis_Select.None;
					
				ENUM_Axis_Select.X:
					IF GV_Axes.bAxisXAllowed THEN
						GV_Axes.eJogAxisSelect:=ENUM_Axis_Select.X;
					END_IF
				
				ENUM_Axis_Select.Y:
					IF GV_Axes.bAxisYAllowed THEN
						GV_Axes.eJogAxisSelect:=ENUM_Axis_Select.Y;
					END_IF
					
				ENUM_Axis_Select.Z:
					IF GV_Axes.bAxisZAllowed THEN
						GV_Axes.eJogAxisSelect:=ENUM_Axis_Select.Z;
					END_IF
					
				ENUM_Axis_Select.Arm:
					IF GV_Axes.bAxisArmAllowed THEN
						GV_Axes.eJogAxisSelect:=ENUM_Axis_Select.Arm;
					END_IF

			END_CASE
		END_IF
	
		IF GV_Axes.eRefAxisRequest<>GV_Axes.eRefAxisSelect THEN 
			CASE GV_Axes.eRefAxisRequest OF

				ENUM_Axis_Select.None:
					GV_Axes.eRefAxisSelect:=ENUM_Axis_Select.None;

				ENUM_Axis_Select.X:
					IF GV_Axes.bReferencingXAllowed THEN
						GV_Axes.eRefAxisSelect:=ENUM_Axis_Select.X;
					END_IF
				
				ENUM_Axis_Select.Y:
					IF GV_Axes.bReferencingYAllowed THEN
						GV_Axes.eRefAxisSelect:=ENUM_Axis_Select.Y;
					END_IF
					
				ENUM_Axis_Select.Z:
					IF GV_Axes.bReferencingZAllowed THEN
						GV_Axes.eRefAxisSelect:=ENUM_Axis_Select.Z;
					END_IF
					
				ENUM_Axis_Select.Arm:
					IF GV_Axes.bReferencingArmAllowed THEN
						GV_Axes.eRefAxisSelect:=ENUM_Axis_Select.Arm;
					END_IF

			END_CASE
		END_IF
	
	(*InProgress*)
		CASE GV_Axes.eJogAxisSelect OF
		
			ENUM_Axis_Select.X:
				IF (NOT GV_General.bSafety) OR (NOT GV_General.bPower) OR (NOT GV_Axes.stAxisX.stDriveAx8206.AxisRef.Status.Operational) OR GV_Axes.stAxisX.bAlAxisFault THEN
					GV_Axes.eJogAxisRequest:=ENUM_Axis_Select.None;
					GV_Axes.eJogAxisSelect:=ENUM_Axis_Select.None;
				END_IF
		
			ENUM_Axis_Select.Y:
				IF (NOT GV_General.bSafety) OR (NOT GV_General.bPower) OR (NOT GV_Axes.stAxisY.stDriveAx8206.AxisRef.Status.Operational) OR GV_Axes.stAxisY.bAlAxisFault THEN
					GV_Axes.eJogAxisRequest:=ENUM_Axis_Select.None;
					GV_Axes.eJogAxisSelect:=ENUM_Axis_Select.None;
				END_IF
				
			ENUM_Axis_Select.Z:
				IF (NOT GV_General.bSafety) OR (NOT GV_General.bPower) OR (NOT GV_Axes.stAxisZ.stDriveAx8206.AxisRef.Status.Operational) OR GV_Axes.stAxisZ.bAlAxisFault OR tonZBrake.Q THEN
					GV_Axes.eJogAxisRequest:=ENUM_Axis_Select.None;
					GV_Axes.eJogAxisSelect:=ENUM_Axis_Select.None;
				END_IF
			
			ENUM_Axis_Select.Arm:
				IF (NOT GV_General.bSafety) OR (NOT GV_General.bPower) OR (NOT GV_Axes.stAxisArm.stDriveAx8206.AxisRef.Status.Operational) OR GV_Axes.stAxisArm.bAlAxisFault THEN
					GV_Axes.eJogAxisRequest:=ENUM_Axis_Select.None;
					GV_Axes.eJogAxisSelect:=ENUM_Axis_Select.None;
				END_IF
			
		END_CASE

		CASE GV_Axes.eRefAxisSelect OF
		
			ENUM_Axis_Select.X:
				IF (NOT GV_General.bSafety) OR (NOT GV_General.bPower) OR (NOT GV_Axes.stAxisX.stDriveAx8206.AxisRef.Status.Operational) OR GV_Axes.stAxisX.bAlAxisFault THEN
					GV_Axes.eRefAxisRequest:=ENUM_Axis_Select.None;
					GV_Axes.eRefAxisSelect:=ENUM_Axis_Select.None;
				END_IF
		
			ENUM_Axis_Select.Y:
				IF (NOT GV_General.bSafety) OR (NOT GV_General.bPower) OR (NOT GV_Axes.stAxisY.stDriveAx8206.AxisRef.Status.Operational) OR GV_Axes.stAxisY.bAlAxisFault THEN
					GV_Axes.eRefAxisRequest:=ENUM_Axis_Select.None;
					GV_Axes.eRefAxisSelect:=ENUM_Axis_Select.None;
				END_IF
				
			ENUM_Axis_Select.Z:
				IF (NOT GV_General.bSafety) OR (NOT GV_General.bPower) OR (NOT GV_Axes.stAxisZ.stDriveAx8206.AxisRef.Status.Operational) OR GV_Axes.stAxisZ.bAlAxisFault THEN
					GV_Axes.eRefAxisRequest:=ENUM_Axis_Select.None;
					GV_Axes.eRefAxisSelect:=ENUM_Axis_Select.None;
				END_IF
			
			ENUM_Axis_Select.Arm:
				IF (NOT GV_General.bSafety) OR (NOT GV_General.bPower) OR (NOT GV_Axes.stAxisArm.stDriveAx8206.AxisRef.Status.Operational) OR GV_Axes.stAxisArm.bAlAxisFault THEN
					GV_Axes.eRefAxisRequest:=ENUM_Axis_Select.None;
					GV_Axes.eRefAxisSelect:=ENUM_Axis_Select.None;
				END_IF
			
		END_CASE

(** VELOCITY **)
	(*Velocity Axis X*)
		CASE GV_OpMode.eOpMode OF
			
			ENUM_OpMode.NONE:
				GV_Axes.lrVelocityAxisX:=0;
			
			ENUM_OpMode.AUTO:
				IF GV_HMI.stAxes.lrVelocityPourcent>0 AND GV_HMI.stAxes.lrVelocityPourcent<=100 THEN
					GV_Axes.lrVelocityAxisX:=GV_Axes.lrAutoMaxSpeedAxisX*(GV_HMI.stAxes.lrVelocityPourcent/100);
				ELSIF GV_HMI.stAxes.lrVelocityPourcent>100 THEN
					GV_Axes.lrVelocityAxisX:=GV_Axes.lrAutoMaxSpeedAxisX;
				ELSE
					GV_Axes.lrVelocityAxisX:=0;
				END_IF
				IF GV_Axes.lrVelocityAxisX>GV_Axes.lrAutoMaxSpeedAxisX THEN
					GV_Axes.lrVelocityAxisX:=GV_Axes.lrAutoMaxSpeedAxisX;
				END_IF
				
			ENUM_OpMode.MANU:
				IF GV_HMI.stAxes.lrVelocityPourcent>0 AND GV_HMI.stAxes.lrVelocityPourcent<=100 THEN
					GV_Axes.lrVelocityAxisX:=GV_Axes.lrJogMaxSpeedAxisX*(GV_HMI.stAxes.lrVelocityPourcent/100);
				ELSIF GV_HMI.stAxes.lrVelocityPourcent>100 THEN
					GV_Axes.lrVelocityAxisX:=GV_Axes.lrJogMaxSpeedAxisX;
				ELSE
					GV_Axes.lrVelocityAxisX:=0;
				END_IF
				IF GV_Axes.lrVelocityAxisX>GV_Axes.lrJogMaxSpeedAxisX THEN
					GV_Axes.lrVelocityAxisX:=GV_Axes.lrJogMaxSpeedAxisX;
				END_IF
				
			ENUM_OpMode.INIT:
				IF GV_HMI.stAxes.lrVelocityPourcent>0 AND GV_HMI.stAxes.lrVelocityPourcent<=100 THEN
					GV_Axes.lrVelocityAxisX:=GV_Axes.lrAutoMaxSpeedAxisX*(GV_HMI.stAxes.lrVelocityPourcent/100);
				ELSIF GV_HMI.stAxes.lrVelocityPourcent>100 THEN
					GV_Axes.lrVelocityAxisX:=GV_Axes.lrAutoMaxSpeedAxisX;
				ELSE
					GV_Axes.lrVelocityAxisX:=0;
				END_IF
				IF GV_Axes.lrVelocityAxisX>GV_Axes.lrAutoMaxSpeedAxisX THEN
					GV_Axes.lrVelocityAxisX:=GV_Axes.lrAutoMaxSpeedAxisX;
				END_IF
				
		END_CASE
	(*Velocity Axis Y*)
		CASE GV_OpMode.eOpMode OF
			
			ENUM_OpMode.NONE:
				GV_Axes.lrVelocityAxisY:=0;
			
			ENUM_OpMode.AUTO:
				IF GV_HMI.stAxes.lrVelocityPourcent>0 AND GV_HMI.stAxes.lrVelocityPourcent<=100 THEN
					GV_Axes.lrVelocityAxisY:=GV_Axes.lrAutoMaxSpeedAxisY*(GV_HMI.stAxes.lrVelocityPourcent/100);
				ELSIF GV_HMI.stAxes.lrVelocityPourcent>100 THEN
					GV_Axes.lrVelocityAxisY:=GV_Axes.lrAutoMaxSpeedAxisY;
				ELSE
					GV_Axes.lrVelocityAxisY:=0;
				END_IF
				IF GV_Axes.lrVelocityAxisY>GV_Axes.lrAutoMaxSpeedAxisY THEN
					GV_Axes.lrVelocityAxisY:=GV_Axes.lrAutoMaxSpeedAxisY;
				END_IF
				
			ENUM_OpMode.MANU:
				IF GV_HMI.stAxes.lrVelocityPourcent>0 AND GV_HMI.stAxes.lrVelocityPourcent<=100 THEN
					GV_Axes.lrVelocityAxisY:=GV_Axes.lrJogMaxSpeedAxisY*(GV_HMI.stAxes.lrVelocityPourcent/100);
				ELSIF GV_HMI.stAxes.lrVelocityPourcent>100 THEN
					GV_Axes.lrVelocityAxisY:=GV_Axes.lrJogMaxSpeedAxisY;
				ELSE
					GV_Axes.lrVelocityAxisY:=0;
				END_IF
				IF GV_Axes.lrVelocityAxisY>GV_Axes.lrJogMaxSpeedAxisY THEN
					GV_Axes.lrVelocityAxisY:=GV_Axes.lrJogMaxSpeedAxisY;
				END_IF
				
			ENUM_OpMode.INIT:
				IF GV_HMI.stAxes.lrVelocityPourcent>0 AND GV_HMI.stAxes.lrVelocityPourcent<=100 THEN
					GV_Axes.lrVelocityAxisY:=GV_Axes.lrAutoMaxSpeedAxisY*(GV_HMI.stAxes.lrVelocityPourcent/100);
				ELSIF GV_HMI.stAxes.lrVelocityPourcent>100 THEN
					GV_Axes.lrVelocityAxisY:=GV_Axes.lrAutoMaxSpeedAxisY;
				ELSE
					GV_Axes.lrVelocityAxisY:=0;
				END_IF
				IF GV_Axes.lrVelocityAxisY>GV_Axes.lrAutoMaxSpeedAxisY THEN
					GV_Axes.lrVelocityAxisY:=GV_Axes.lrAutoMaxSpeedAxisY;
				END_IF
				
		END_CASE
	(*Velocity Axis Z*)
		CASE GV_OpMode.eOpMode OF
			
			ENUM_OpMode.NONE:
				GV_Axes.lrVelocityAxisZ:=0;
			
			ENUM_OpMode.AUTO:
				IF GV_HMI.stAxes.lrVelocityPourcent>0 AND GV_HMI.stAxes.lrVelocityPourcent<=100 THEN
					GV_Axes.lrVelocityAxisZ:=GV_Axes.lrAutoMaxSpeedAxisZ*(GV_HMI.stAxes.lrVelocityPourcent/100);
				ELSIF GV_HMI.stAxes.lrVelocityPourcent>100 THEN
					GV_Axes.lrVelocityAxisZ:=GV_Axes.lrAutoMaxSpeedAxisZ;
				ELSE
					GV_Axes.lrVelocityAxisZ:=0;
				END_IF
				IF GV_Axes.lrVelocityAxisZ>GV_Axes.lrAutoMaxSpeedAxisZ THEN
					GV_Axes.lrVelocityAxisZ:=GV_Axes.lrAutoMaxSpeedAxisZ;
				END_IF
				
			ENUM_OpMode.MANU:
				IF GV_HMI.stAxes.lrVelocityPourcent>0 AND GV_HMI.stAxes.lrVelocityPourcent<=100 THEN
					GV_Axes.lrVelocityAxisZ:=GV_Axes.lrJogMaxSpeedAxisZ*(GV_HMI.stAxes.lrVelocityPourcent/100);
				ELSIF GV_HMI.stAxes.lrVelocityPourcent>100 THEN
					GV_Axes.lrVelocityAxisZ:=GV_Axes.lrJogMaxSpeedAxisZ;
				ELSE
					GV_Axes.lrVelocityAxisZ:=0;
				END_IF
				IF GV_Axes.lrVelocityAxisZ>GV_Axes.lrJogMaxSpeedAxisZ THEN
					GV_Axes.lrVelocityAxisZ:=GV_Axes.lrJogMaxSpeedAxisZ;
				END_IF
				
			ENUM_OpMode.INIT:
				IF GV_HMI.stAxes.lrVelocityPourcent>0 AND GV_HMI.stAxes.lrVelocityPourcent<=100 THEN
					GV_Axes.lrVelocityAxisZ:=GV_Axes.lrAutoMaxSpeedAxisZ*(GV_HMI.stAxes.lrVelocityPourcent/100);
				ELSIF GV_HMI.stAxes.lrVelocityPourcent>100 THEN
					GV_Axes.lrVelocityAxisZ:=GV_Axes.lrAutoMaxSpeedAxisZ;
				ELSE
					GV_Axes.lrVelocityAxisZ:=0;
				END_IF
				IF GV_Axes.lrVelocityAxisZ>GV_Axes.lrAutoMaxSpeedAxisZ THEN
					GV_Axes.lrVelocityAxisZ:=GV_Axes.lrAutoMaxSpeedAxisZ;
				END_IF
				
		END_CASE
	(*Velocity Axis Arm*)
		CASE GV_OpMode.eOpMode OF
			
			ENUM_OpMode.NONE:
				GV_Axes.lrVelocityAxisArm:=0;
			
			ENUM_OpMode.AUTO:
				IF GV_HMI.stAxes.lrVelocityPourcent>0 AND GV_HMI.stAxes.lrVelocityPourcent<=100 THEN
					GV_Axes.lrVelocityAxisArm:=GV_Axes.lrAutoMaxSpeedAxisArm*(GV_HMI.stAxes.lrVelocityPourcent/100);
				ELSIF GV_HMI.stAxes.lrVelocityPourcent>100 THEN
					GV_Axes.lrVelocityAxisArm:=GV_Axes.lrAutoMaxSpeedAxisArm;
				ELSE
					GV_Axes.lrVelocityAxisArm:=0;
				END_IF
				IF GV_Axes.lrVelocityAxisArm>GV_Axes.lrAutoMaxSpeedAxisArm THEN
					GV_Axes.lrVelocityAxisArm:=GV_Axes.lrAutoMaxSpeedAxisArm;
				END_IF
				
			ENUM_OpMode.MANU:
				IF GV_HMI.stAxes.lrVelocityPourcent>0 AND GV_HMI.stAxes.lrVelocityPourcent<=100 THEN
					GV_Axes.lrVelocityAxisArm:=GV_Axes.lrJogMaxSpeedAxisArm*(GV_HMI.stAxes.lrVelocityPourcent/100);
				ELSIF GV_HMI.stAxes.lrVelocityPourcent>100 THEN
					GV_Axes.lrVelocityAxisArm:=GV_Axes.lrJogMaxSpeedAxisArm;
				ELSE
					GV_Axes.lrVelocityAxisArm:=0;
				END_IF
				IF GV_Axes.lrVelocityAxisArm>GV_Axes.lrJogMaxSpeedAxisArm THEN
					GV_Axes.lrVelocityAxisArm:=GV_Axes.lrJogMaxSpeedAxisArm;
				END_IF
				
			ENUM_OpMode.INIT:
				IF GV_HMI.stAxes.lrVelocityPourcent>0 AND GV_HMI.stAxes.lrVelocityPourcent<=100 THEN
					GV_Axes.lrVelocityAxisArm:=GV_Axes.lrAutoMaxSpeedAxisArm*(GV_HMI.stAxes.lrVelocityPourcent/100);
				ELSIF GV_HMI.stAxes.lrVelocityPourcent>100 THEN
					GV_Axes.lrVelocityAxisArm:=GV_Axes.lrAutoMaxSpeedAxisArm;
				ELSE
					GV_Axes.lrVelocityAxisArm:=0;
				END_IF
				IF GV_Axes.lrVelocityAxisArm>GV_Axes.lrAutoMaxSpeedAxisArm THEN
					GV_Axes.lrVelocityAxisArm:=GV_Axes.lrAutoMaxSpeedAxisArm;
				END_IF
				
		END_CASE

(** AXIS X **)
	(* Setup *)
		GV_Axes.stAxisX.bPresence:=TRUE; // Axis Presence
		fbEventGroupAssignement(iEventGroup:=GV_Axes.stAxisX.iEventGroup);
		GV_Axes.stAxisX.strIdHMI:='X'; // String for events on HMI
		GV_Axes.stAxisX.iIdHMI:=UDINT_TO_INT(GV_Axes.stAxisX.stDriveAx8206.AxisRef.NcToPlc.AxisId); // Number for events on HMI
		(*Power*)
			IF ((GV_General.bSafety AND GV_General.bPower AND (NOT GV_Axes.stAxisX.bAlAxisFault)) OR (GV_Axes.stAxisX.bPowerEnable AND ((GV_Axes.stAxisX.bStopExecute AND (NOT GV_Axes.stAxisX.bStopDone))) OR ((GV_Axes.stAxisX.bHaltExecute AND (NOT GV_Axes.stAxisX.bHaltDone))))) AND (NOT GV_General.bRebootRequest) AND (NOT GV_General.bShutdownRequest) THEN
				GV_Axes.stAxisX.bPowerEnable:=TRUE;
			ELSE
				GV_Axes.stAxisX.bPowerEnable:=FALSE;
			END_IF
		(*Stop*)
			GV_Axes.stAxisX.bStopExecute:=(NOT GV_General.bSafety) OR (NOT GV_General.bPower) OR GV_General.bRebootRequest OR GV_General.bShutdownRequest (*OR (GV_OpMode.eOpMode=ENUM_OpMode.AUTO AND GV_Cycle.bCycleInProgress AND (NOT GV_Cycle.bStartStop))*); // Have to stop
		(*Halt*)
			GV_Axes.stAxisX.bHaltExecute:=(GV_OpMode.eOpMode=ENUM_OpMode.AUTO AND GV_Cycle.bCycleInProgress AND (NOT GV_Cycle.bStartStop)); // Have to halt
		(*Abort*)
			//GV_Axes.stAxisX.bAbort:=(NOT GV_Axes.stAxisX.stDriveAx8206.AxisRef.Status.NotMoving) AND (GV_OpMode.eOpMode=ENUM_OpMode.AUTO AND GV_Cycle.bCycleInProgress AND (NOT GV_Cycle.bStartStop)); // Have to abort
		(*Reset*)
			GV_Axes.stAxisX.bEventAck:=GV_HMI.bEventAck; // Events Acknowledgement	
		(*Jog*)
			GV_Axes.stAxisX.bJogEnable:=GV_OpMode.eOpMode=ENUM_OpMode.MANU AND GV_Axes.stAxisX.stDriveAx8206.AxisRef.Status.Operational AND (NOT GV_Axes.stAxisX.bAlAxisFault) AND
			((GV_Handwheel.aId[1].bEnable AND GV_Handwheel.aId[1].eAxisSelect=ENUM_Axis_Select.X) OR ((NOT GV_Handwheel.aId[1].bEnable) AND GV_HMI.iCurrentScreenNumber=210 AND GV_Axes.eJogAxisSelect=ENUM_Axis_Select.X));
			IF GV_Axes.stAxisX.bJogEnable AND (NOT GV_Handwheel.aId[1].bEnable) THEN // Jog from HMI
				GV_Axes.stAxisX.eJogMode:=TC2_MC2.E_JogMode.MC_JOGMODE_CONTINOUS; // Jog Mode
				GV_Axes.stAxisX.bJogPlus:=GV_HMI.stAxes.bButtonPlus; // Jog +
				GV_Axes.stAxisX.bJogMinus:=GV_HMI.stAxes.bButtonMinus; // Jog -
				GV_Axes.stAxisX.lrJogPos:=0; // Jog Position -> Only in mode INCHING
				GV_Axes.stAxisX.lrJogVel:=GV_Axes.lrVelocityAxisX; // Jog Velocity
				GV_Axes.stAxisX.lrJogAcc:=0; // Jog Acceleration -> see the Axis Configuration in the System Manager
				GV_Axes.stAxisX.lrJogDec:=0; // Jog Decelration -> see the Axis Configuration in the System Manager
				GV_Axes.stAxisX.lrJogJerk:=0; // Jog Jerk -> see the Axis Configuration in the System Manager
			ELSIF GV_Axes.stAxisX.bJogEnable AND GV_Handwheel.aId[1].bEnable (*AND GV_Handwheel.aId[1].eJogMode=ENUM_Jog_Mode.Inching*) AND GV_Handwheel.aId[1].bJogRequestRisingEdge THEN // Incremental from Handwheel
				GV_Axes.stAxisX.eJogMode:=TC2_MC2.E_JogMode.MC_JOGMODE_INCHING; // Jog Mode
				GV_Axes.stAxisX.bJogPlus:=(GV_Handwheel.aId[1].eJogDirection=ENUM_Jog_Direction.Plus); // Incr +
				GV_Axes.stAxisX.bJogMinus:=(GV_Handwheel.aId[1].eJogDirection=ENUM_Jog_Direction.Minus); // Incr -
				GV_Axes.stAxisX.lrJogPos:=GV_Handwheel.aId[1].lrJogIncrRequest; // Jog Position
				GV_Axes.stAxisX.lrJogVel:=GV_Axes.lrJogMaxSpeedAxisX;//GV_Axes.lrVelocityAxisX; // Jog Velocity
				GV_Axes.stAxisX.lrJogAcc:=0; // Jog Acceleration -> see the Axis Configuration in the System Manager
				GV_Axes.stAxisX.lrJogDec:=0; // Jog Decelration -> see the Axis Configuration in the System Manager
				GV_Axes.stAxisX.lrJogJerk:=0; // Jog Jerk -> see the Axis Configuration in the System Manager
// 			ELSIF GV_Axes.stAxisX.bJogEnable AND GV_Handwheel.aId[1].bEnable AND GV_Handwheel.aId[1].eJogMode=ENUM_Jog_Mode.Continous AND GV_Handwheel.aId[1].bJogRequestRisingEdge THEN // Jog from Handwheel button only
// 				GV_Axes.stAxisX.eJogMode:=TC2_MC2.E_JogMode.MC_JOGMODE_CONTINOUS; // Jog Mode
// 				GV_Axes.stAxisX.bJogPlus:=(GV_Handwheel.aId[1].eJogDirection=ENUM_Jog_Direction.Plus); // Jog +
// 				GV_Axes.stAxisX.bJogMinus:=(GV_Handwheel.aId[1].eJogDirection=ENUM_Jog_Direction.Minus); // Jog -
// 				GV_Axes.stAxisX.lrJogPos:=0; // Jog Position -> Only in mode INCHING
// 				GV_Axes.stAxisX.lrJogVel:=GV_Axes.lrVelocityAxisX; // Jog Velocity
// 				GV_Axes.stAxisX.lrJogAcc:=0; // Jog Acceleration -> see the Axis Configuration in the System Manager
// 				GV_Axes.stAxisX.lrJogDec:=0; // Jog Decelration -> see the Axis Configuration in the System Manager
// 				GV_Axes.stAxisX.lrJogJerk:=0; // Jog Jerk -> see the Axis Configuration in the System Manager
			ELSE
				GV_Axes.stAxisX.bJogPlus:=FALSE; // Jog +
				GV_Axes.stAxisX.bJogMinus:=FALSE; // Jog -
				GV_Axes.stAxisX.lrJogPos:=0; // Jog Position
				GV_Axes.stAxisX.lrJogVel:=0; // Jog Velocity
				GV_Axes.stAxisX.lrJogAcc:=0; // Jog Acceleration -> see the Axis Configuration in the System Manager
				GV_Axes.stAxisX.lrJogDec:=0; // Jog Decelration -> see the Axis Configuration in the System Manager
				GV_Axes.stAxisX.lrJogJerk:=0; // Jog Jerk -> see the Axis Configuration in the System Manager				
			END_IF
		(*AUTO*)
			GV_Axes.stAxisX.bAutoEnable:=GV_OpMode.eOpMode=ENUM_OpMode.AUTO AND GV_Cycle.bStartStop AND GV_Axes.stAxisX.stDriveAx8206.AxisRef.Status.Operational AND (NOT GV_Axes.stAxisX.bAlAxisFault);
			IF  GV_Axes.stAxisX.bAutoEnable THEN
				GV_Axes.stAxisX.lrAutoVelAbs:=GV_Axes.lrVelocityAxisX; // AUTO Velocity
				GV_Axes.stAxisX.lrAutoAccAbs:=0; // AUTO Acceleration -> see the Axis Configuration in the System Manager
				GV_Axes.stAxisX.lrAutoDecAbs:=0; // AUTO Decelration -> see the Axis Configuration in the System Manager
				GV_Axes.stAxisX.lrAutoJerkAbs:=0; // AUTO Jerk -> see the Axis Configuration in the System Manager
			ELSE
				GV_Axes.stAxisX.lrAutoVelAbs:=0; // AUTO Velocity
				GV_Axes.stAxisX.lrAutoAccAbs:=0; // AUTO Acceleration -> see the Axis Configuration in the System Manager
				GV_Axes.stAxisX.lrAutoDecAbs:=0; // AUTO Decelration -> see the Axis Configuration in the System Manager
				GV_Axes.stAxisX.lrAutoJerkAbs:=0; // AUTO Jerk -> see the Axis Configuration in the System Manager
			END_IF
		(*Referencing*)
			GV_Axes.stAxisX.bSetOffsetExecute:=GV_OpMode.eOpMode=ENUM_OpMode.MANU AND GV_Axes.stAxisX.stDriveAx8206.AxisRef.Status.Operational AND (NOT GV_Axes.stAxisX.bAlAxisFault) AND GV_HMI.iCurrentScreenNumber=308 AND GV_Axes.eRefAxisSelect=ENUM_Axis_Select.X AND GV_HMI.stAxes.rtButtonReferencingAxis.Q;
			GV_Axes.stAxisX.bDeleteOffsetExecute:=FALSE; // Not used in the HMI, we can use it from here or add it in the HMI later if it's necessary
		(*ReadParameter BOOL*)
			GV_Axes.stAxisX.bReadbEnable:=(GV_Axes.stAxisX.mcAxisReadParameterb=MC_AxisParameter.AxisEnMinSoftPosLimit OR GV_Axes.stAxisX.mcAxisReadParameterb=MC_AxisParameter.AxisEnMaxSoftPosLimit) AND GV_Axes.stAxisX.stDriveAx8206.AxisRef.Status.Operational;
			IF GV_Axes.stAxisX.stDriveAx8206.AxisRef.Status.Operational THEN
				IF GV_Axes.stAxisX.mcAxisReadParameterb=MC_AxisParameter.AxisEnMaxSoftPosLimit THEN
					IF GV_General.bIsBlinking05s THEN
						GV_Axes.stAxisX.mcAxisReadParameterb:=MC_AxisParameter.AxisEnMinSoftPosLimit;
					ELSE
						IF GV_Axes.stAxisX.bReadbValid THEN
							GV_Axes.stAxisX.bReadEnMaxSoftPosLimit:=GV_Axes.stAxisX.bReadbValue;
						END_IF
					END_IF
				ELSIF GV_Axes.stAxisX.mcAxisReadParameterb=MC_AxisParameter.AxisEnMinSoftPosLimit THEN
					IF GV_General.bIsBlinking05s THEN
						GV_Axes.stAxisX.mcAxisReadParameterb:=MC_AxisParameter.AxisEnMaxSoftPosLimit;
					ELSE
						IF GV_Axes.stAxisX.bReadbValid THEN
							GV_Axes.stAxisX.bReadEnMinSoftPosLimit:=GV_Axes.stAxisX.bReadbValue;
						END_IF
					END_IF
				ELSE
					GV_Axes.stAxisX.mcAxisReadParameterb:=MC_AxisParameter.AxisEnMinSoftPosLimit;
				END_IF
			END_IF
		(*ReadParameter LREAL*)
			GV_Axes.stAxisX.bReadlrEnable:=(GV_Axes.stAxisX.mcAxisReadParameterlr=MC_AxisParameter.AxisMinSoftPosLimit OR GV_Axes.stAxisX.mcAxisReadParameterlr=MC_AxisParameter.AxisMaxSoftPosLimit) AND GV_Axes.stAxisX.stDriveAx8206.AxisRef.Status.Operational;
			IF GV_Axes.stAxisX.stDriveAx8206.AxisRef.Status.Operational THEN
				IF GV_Axes.stAxisX.mcAxisReadParameterlr=MC_AxisParameter.AxisMaxSoftPosLimit THEN
					IF GV_General.bIsBlinking05s THEN
						GV_Axes.stAxisX.mcAxisReadParameterlr:=MC_AxisParameter.AxisMinSoftPosLimit;
					ELSE
						IF GV_Axes.stAxisX.bReadlrValid THEN
							GV_Axes.stAxisX.lrReadMaxSoftPosLimit:=GV_Axes.stAxisX.lrReadlrValue;
						END_IF
					END_IF
				ELSIF GV_Axes.stAxisX.mcAxisReadParameterlr=MC_AxisParameter.AxisMinSoftPosLimit THEN
					IF (NOT GV_General.bIsBlinking05s) THEN
						GV_Axes.stAxisX.mcAxisReadParameterlr:=MC_AxisParameter.AxisMaxSoftPosLimit;
					ELSE
						IF GV_Axes.stAxisX.bReadlrValid THEN
							GV_Axes.stAxisX.lrReadMinSoftPosLimit:=GV_Axes.stAxisX.lrReadlrValue;
						END_IF
					END_IF
				ELSE
					GV_Axes.stAxisX.mcAxisReadParameterlr:=MC_AxisParameter.AxisMinSoftPosLimit;
				END_IF
			END_IF	
		(*WriteParameter BOOL*)
			GV_Axes.stAxisX.bWritebExecute:=GV_Axes.eRefAxisSelect=ENUM_Axis_Select.X AND (GV_HMI.stAxes.rtButtonMinSofltLimit.Q OR GV_HMI.stAxes.rtButtonMaxSofltLimit.Q) AND GV_Axes.stAxisX.stDriveAx8206.AxisRef.Status.Operational;
			IF GV_Axes.stAxisX.stDriveAx8206.AxisRef.Status.Operational AND (NOT GV_Axes.stAxisX.stDriveAx8206.AxisRef.Status.Moving) THEN
				IF GV_HMI.stAxes.rtButtonMinSofltLimit.Q THEN
					GV_Axes.stAxisX.mcAxisWriteParameterb:=MC_AxisParameter.AxisEnMinSoftPosLimit;
					IF GV_Axes.stAxisX.bReadEnMinSoftPosLimit THEN
						GV_Axes.stAxisX.bWritebValue:=FALSE;
					ELSE
						GV_Axes.stAxisX.bWritebValue:=TRUE;
					END_IF
				ELSIF GV_HMI.stAxes.rtButtonMaxSofltLimit.Q THEN
					GV_Axes.stAxisX.mcAxisWriteParameterb:=MC_AxisParameter.AxisEnMaxSoftPosLimit;
					IF GV_Axes.stAxisX.bReadEnMaxSoftPosLimit THEN
						GV_Axes.stAxisX.bWritebValue:=FALSE;
					ELSE
						GV_Axes.stAxisX.bWritebValue:=TRUE;
					END_IF
				END_IF
			END_IF
		(*WriteParameter LREAL*)
// 			bAxisXWrite1:=FALSE;
// 			bAxisXWrite2:=FALSE;
// 			bAxisXWrite3:=FALSE;
// 			bAxisXWrite4:=FALSE;
// 			IF GV_Tool_Magazine.stManipulator.ePositionMag=ENUM_Position_Magazine.Top THEN
// 				IF GV_Tool_Magazine.stManipulator.lrXPosition<>GV_Tool_Magazine.stManipulator.lrXTunnel THEN
// 					GV_Axes.stAxisX.lrValueMax:=-10;
// 					GV_Axes.stAxisX.lrValueMin:=-350;
// 					bAxisXWrite1:=TRUE;
// 				ELSE
// 					GV_Axes.stAxisX.lrValueMax:=-10;
// 					GV_Axes.stAxisX.lrValueMin:=-800;
// 					bAxisXWrite2:=TRUE;
// 				END_IF
// 			END_IF
// 			IF GV_Tool_Magazine.stManipulator.ePositionMag=ENUM_Position_Magazine.Bottom THEN
// 				IF GV_Tool_Magazine.stManipulator.lrXPosition<>GV_Tool_Magazine.stManipulator.lrXTunnel THEN
// 					GV_Axes.stAxisX.lrValueMax:=-450;
// 					GV_Axes.stAxisX.lrValueMin:=-800;
// 					bAxisXWrite3:=TRUE;
// 				ELSE
// 					GV_Axes.stAxisX.lrValueMax:=-10;
// 					GV_Axes.stAxisX.lrValueMin:=-800;
// 					bAxisXWrite4:=TRUE;
// 				END_IF
// 			END_IF
// 			rtAxisXWrite1(CLK:=bAxisXWrite1);
// 			rtAxisXWrite2(CLK:=bAxisXWrite2);
// 			rtAxisXWrite3(CLK:=bAxisXWrite3);
// 			rtAxisXWrite4(CLK:=bAxisXWrite4);
// 			IF rtAxisXWrite1.Q OR rtAxisXWrite2.Q OR rtAxisXWrite3.Q OR rtAxisXWrite4.Q THEN
// 				GV_Axes.stAxisX.mcAxisWriteParameterlr:=MC_AxisParameter.AxisMaxSoftPosLimit;
// 				GV_Axes.stAxisX.lrWritelrValue:=GV_Axes.stAxisX.lrValueMax;
// 				bAxisXWriteMin:=FALSE;
// 				bAxisXWriteMax:=TRUE;
// 			END_IF
// 			IF bAxisXWriteMax AND GV_Axes.stAxisX.bWritelrBusy THEN
// 				GV_Axes.stAxisX.mcAxisWriteParameterlr:=MC_AxisParameter.AxisMinSoftPosLimit;
// 				GV_Axes.stAxisX.lrWritelrValue:=GV_Axes.stAxisX.lrValueMin;
// 				bAxisXWriteMin:=TRUE;
// 				bAxisXWriteMax:=FALSE;
// 			END_IF
// 			IF bAxisXWriteMin AND GV_Axes.stAxisX.bWritelrBusy THEN
// 				bAxisXWriteMin:=FALSE;
// 				bAxisXWriteMax:=FALSE;
// 			END_IF
// 			GV_Axes.stAxisX.bWritelrExecute:=(bAxisXWriteMax OR bAxisXWriteMin) AND GV_Axes.stAxisX.bWritelrDone AND (NOT GV_Axes.stAxisX.bWritelrBusy) AND GV_Axes.stAxisX.stDriveAx8206.AxisRef.Status.Operational;
// 			
	(* Fb *)
		IF GV_Axes.stAxisX.bPresence THEN
			fbAxisX(
					stAxis:=GV_Axes.stAxisX,
					);
		END_IF

(** AXIS Y **)
	(* Setup *)
		GV_Axes.stAxisY.bPresence:=TRUE; // Axis Presence
		fbEventGroupAssignement(iEventGroup:=GV_Axes.stAxisY.iEventGroup);
		GV_Axes.stAxisY.strIdHMI:='Y'; // String for events on HMI
		GV_Axes.stAxisY.iIdHMI:=UDINT_TO_INT(GV_Axes.stAxisY.stDriveAx8206.AxisRef.NcToPlc.AxisId); // Number for events on HMI
		(*Power*)
			IF ((GV_General.bSafety AND GV_General.bPower AND (NOT GV_Axes.stAxisY.bAlAxisFault)) OR (GV_Axes.stAxisY.bPowerEnable AND ((GV_Axes.stAxisY.bStopExecute AND (NOT GV_Axes.stAxisY.bStopDone))) OR ((GV_Axes.stAxisY.bHaltExecute AND (NOT GV_Axes.stAxisY.bHaltDone))))) AND (NOT GV_General.bRebootRequest) AND (NOT GV_General.bShutdownRequest) THEN
				GV_Axes.stAxisY.bPowerEnable:=TRUE;
			ELSE
				GV_Axes.stAxisY.bPowerEnable:=FALSE;
			END_IF
		(*Stop*)
			GV_Axes.stAxisY.bStopExecute:=(NOT GV_General.bSafety) OR (NOT GV_General.bPower) OR GV_General.bRebootRequest OR GV_General.bShutdownRequest (*OR (GV_OpMode.eOpMode=ENUM_OpMode.AUTO AND GV_Cycle.bCycleInProgress AND (NOT GV_Cycle.bStartStop))*); // Have to stop
		(*Halt*)
			GV_Axes.stAxisY.bHaltExecute:=(GV_OpMode.eOpMode=ENUM_OpMode.AUTO AND GV_Cycle.bCycleInProgress AND (NOT GV_Cycle.bStartStop)); // Have to halt
		(*Abort*)
			//GV_Axes.stAxisY.bAbort:=(NOT GV_Axes.stAxisY.stDriveAx8206.AxisRef.Status.NotMoving) AND (GV_OpMode.eOpMode=ENUM_OpMode.AUTO AND GV_Cycle.bCycleInProgress AND (NOT GV_Cycle.bStartStop)); // Have to abort
		(*Reset*)
			GV_Axes.stAxisY.bEventAck:=GV_HMI.bEventAck; // Events Acknowledgement	
		(*Jog*)
			GV_Axes.stAxisY.bJogEnable:=GV_OpMode.eOpMode=ENUM_OpMode.MANU AND GV_Axes.stAxisY.stDriveAx8206.AxisRef.Status.Operational AND (NOT GV_Axes.stAxisY.bAlAxisFault) AND
			((GV_Handwheel.aId[1].bEnable AND GV_Handwheel.aId[1].eAxisSelect=ENUM_Axis_Select.Y) OR ((NOT GV_Handwheel.aId[1].bEnable) AND GV_HMI.iCurrentScreenNumber=210 AND GV_Axes.eJogAxisSelect=ENUM_Axis_Select.Y));
			IF GV_Axes.stAxisY.bJogEnable AND (NOT GV_Handwheel.aId[1].bEnable) THEN // Jog from HMI
				GV_Axes.stAxisY.eJogMode:=TC2_MC2.E_JogMode.MC_JOGMODE_CONTINOUS; // Jog Mode
				GV_Axes.stAxisY.bJogPlus:=GV_HMI.stAxes.bButtonPlus; // Jog +
				GV_Axes.stAxisY.bJogMinus:=GV_HMI.stAxes.bButtonMinus; // Jog -
				GV_Axes.stAxisY.lrJogPos:=0; // Jog Position -> Only in mode INCHING
				GV_Axes.stAxisY.lrJogVel:=GV_Axes.lrVelocityAxisY; // Jog Velocity
				GV_Axes.stAxisY.lrJogAcc:=0; // Jog Acceleration -> see the Axis Configuration in the System Manager
				GV_Axes.stAxisY.lrJogDec:=0; // Jog Decelration -> see the Axis Configuration in the System Manager
				GV_Axes.stAxisY.lrJogJerk:=0; // Jog Jerk -> see the Axis Configuration in the System Manager
			ELSIF GV_Axes.stAxisY.bJogEnable AND GV_Handwheel.aId[1].bEnable AND GV_Handwheel.aId[1].bJogRequestRisingEdge THEN // Jog from Handwheel
				GV_Axes.stAxisY.eJogMode:=TC2_MC2.E_JogMode.MC_JOGMODE_INCHING; // Jog Mode
				GV_Axes.stAxisY.bJogPlus:=(GV_Handwheel.aId[1].eJogDirection=ENUM_Jog_Direction.Plus); // Jog +
				GV_Axes.stAxisY.bJogMinus:=(GV_Handwheel.aId[1].eJogDirection=ENUM_Jog_Direction.Minus); // Jog -
				GV_Axes.stAxisY.lrJogPos:=GV_Handwheel.aId[1].lrJogIncrRequest; // Jog Position
				GV_Axes.stAxisY.lrJogVel:=GV_Axes.lrJogMaxSpeedAxisY;//GV_Axes.lrVelocityAxisY; // Jog Velocity
				GV_Axes.stAxisY.lrJogAcc:=0; // Jog Acceleration -> see the Axis Configuration in the System Manager
				GV_Axes.stAxisY.lrJogDec:=0; // Jog Decelration -> see the Axis Configuration in the System Manager
				GV_Axes.stAxisY.lrJogJerk:=0; // Jog Jerk -> see the Axis Configuration in the System Manager
			ELSE
				GV_Axes.stAxisY.bJogPlus:=FALSE; // Jog +
				GV_Axes.stAxisY.bJogMinus:=FALSE; // Jog -
				GV_Axes.stAxisY.lrJogPos:=0; // Jog Position
				GV_Axes.stAxisY.lrJogVel:=0; // Jog Velocity
				GV_Axes.stAxisY.lrJogAcc:=0; // Jog Acceleration -> see the Axis Configuration in the System Manager
				GV_Axes.stAxisY.lrJogDec:=0; // Jog Decelration -> see the Axis Configuration in the System Manager
				GV_Axes.stAxisY.lrJogJerk:=0; // Jog Jerk -> see the Axis Configuration in the System Manager				
			END_IF
		(*AUTO*)
			GV_Axes.stAxisY.bAutoEnable:=GV_OpMode.eOpMode=ENUM_OpMode.AUTO AND GV_Cycle.bStartStop AND GV_Axes.stAxisY.stDriveAx8206.AxisRef.Status.Operational AND (NOT GV_Axes.stAxisY.bAlAxisFault);
			IF  GV_Axes.stAxisY.bAutoEnable THEN
				GV_Axes.stAxisY.lrAutoVelAbs:=GV_Axes.lrVelocityAxisY; // AUTO Velocity
				GV_Axes.stAxisY.lrAutoAccAbs:=0; // AUTO Acceleration -> see the Axis Configuration in the System Manager
				GV_Axes.stAxisY.lrAutoDecAbs:=0; // AUTO Decelration -> see the Axis Configuration in the System Manager
				GV_Axes.stAxisY.lrAutoJerkAbs:=0; // AUTO Jerk -> see the Axis Configuration in the System Manager
			ELSE
				GV_Axes.stAxisY.lrAutoVelAbs:=0; // AUTO Velocity
				GV_Axes.stAxisY.lrAutoAccAbs:=0; // AUTO Acceleration -> see the Axis Configuration in the System Manager
				GV_Axes.stAxisY.lrAutoDecAbs:=0; // AUTO Decelration -> see the Axis Configuration in the System Manager
				GV_Axes.stAxisY.lrAutoJerkAbs:=0; // AUTO Jerk -> see the Axis Configuration in the System Manager
			END_IF
		(*Referencing*)
			GV_Axes.stAxisY.bSetOffsetExecute:=GV_OpMode.eOpMode=ENUM_OpMode.MANU AND GV_Axes.stAxisY.stDriveAx8206.AxisRef.Status.Operational AND (NOT GV_Axes.stAxisY.bAlAxisFault) AND GV_HMI.iCurrentScreenNumber=308 AND GV_Axes.eRefAxisSelect=ENUM_Axis_Select.Y AND GV_HMI.stAxes.rtButtonReferencingAxis.Q;
			GV_Axes.stAxisY.bDeleteOffsetExecute:=FALSE; // Not used in the HMI, we can use it from here or add it in the HMI later if it's necessary
		(*ReadParameter BOOL*)
			GV_Axes.stAxisY.bReadbEnable:=(GV_Axes.stAxisY.mcAxisReadParameterb=MC_AxisParameter.AxisEnMinSoftPosLimit OR GV_Axes.stAxisY.mcAxisReadParameterb=MC_AxisParameter.AxisEnMaxSoftPosLimit) AND GV_Axes.stAxisY.stDriveAx8206.AxisRef.Status.Operational;
			IF GV_Axes.stAxisY.stDriveAx8206.AxisRef.Status.Operational THEN
				IF GV_Axes.stAxisY.mcAxisReadParameterb=MC_AxisParameter.AxisEnMaxSoftPosLimit THEN
					IF GV_General.bIsBlinking05s THEN
						GV_Axes.stAxisY.mcAxisReadParameterb:=MC_AxisParameter.AxisEnMinSoftPosLimit;
					ELSE
						IF GV_Axes.stAxisY.bReadbValid THEN
							GV_Axes.stAxisY.bReadEnMaxSoftPosLimit:=GV_Axes.stAxisY.bReadbValue;
						END_IF
					END_IF
				ELSIF GV_Axes.stAxisY.mcAxisReadParameterb=MC_AxisParameter.AxisEnMinSoftPosLimit THEN
					IF GV_General.bIsBlinking05s THEN
						GV_Axes.stAxisY.mcAxisReadParameterb:=MC_AxisParameter.AxisEnMaxSoftPosLimit;
					ELSE
						IF GV_Axes.stAxisY.bReadbValid THEN
							GV_Axes.stAxisY.bReadEnMinSoftPosLimit:=GV_Axes.stAxisY.bReadbValue;
						END_IF
					END_IF
				ELSE
					GV_Axes.stAxisY.mcAxisReadParameterb:=MC_AxisParameter.AxisEnMinSoftPosLimit;
				END_IF
			END_IF
		(*ReadParameter LREAL*)
			GV_Axes.stAxisY.bReadlrEnable:=(GV_Axes.stAxisY.mcAxisReadParameterlr=MC_AxisParameter.AxisMinSoftPosLimit OR GV_Axes.stAxisY.mcAxisReadParameterlr=MC_AxisParameter.AxisMaxSoftPosLimit) AND GV_Axes.stAxisY.stDriveAx8206.AxisRef.Status.Operational;
			IF GV_Axes.stAxisY.stDriveAx8206.AxisRef.Status.Operational THEN
				IF GV_Axes.stAxisY.mcAxisReadParameterlr=MC_AxisParameter.AxisMaxSoftPosLimit THEN
					IF GV_General.bIsBlinking05s THEN
						GV_Axes.stAxisY.mcAxisReadParameterlr:=MC_AxisParameter.AxisMinSoftPosLimit;
					ELSE
						IF GV_Axes.stAxisY.bReadlrValid THEN
							GV_Axes.stAxisY.lrReadMaxSoftPosLimit:=GV_Axes.stAxisY.lrReadlrValue;
						END_IF
					END_IF
				ELSIF GV_Axes.stAxisY.mcAxisReadParameterlr=MC_AxisParameter.AxisMinSoftPosLimit THEN
					IF (NOT GV_General.bIsBlinking05s) THEN
						GV_Axes.stAxisY.mcAxisReadParameterlr:=MC_AxisParameter.AxisMaxSoftPosLimit;
					ELSE
						IF GV_Axes.stAxisY.bReadlrValid THEN
							GV_Axes.stAxisY.lrReadMinSoftPosLimit:=GV_Axes.stAxisY.lrReadlrValue;
						END_IF
					END_IF
				ELSE
					GV_Axes.stAxisY.mcAxisReadParameterlr:=MC_AxisParameter.AxisMinSoftPosLimit;
				END_IF
			END_IF	
		(*WriteParameter BOOL*)
// 			GV_Axes.stAxisY.bWritebExecute:=GV_Axes.eRefAxisSelect=ENUM_Axis_Select.Y AND (GV_HMI.stAxes.rtButtonMinSofltLimit.Q OR GV_HMI.stAxes.rtButtonMaxSofltLimit.Q) AND GV_Axes.stAxisY.stDriveAx8206.AxisRef.Status.Operational;
// 			IF GV_Axes.stAxisY.stDriveAx8206.AxisRef.Status.Operational AND (NOT GV_Axes.stAxisY.stDriveAx8206.AxisRef.Status.Moving) THEN
// 				IF GV_HMI.stAxes.rtButtonMinSofltLimit.Q THEN
// 					GV_Axes.stAxisY.mcAxisWriteParameterb:=MC_AxisParameter.AxisEnMinSoftPosLimit;
// 					IF GV_Axes.stAxisY.bReadEnMinSoftPosLimit THEN
// 						GV_Axes.stAxisY.bWritebValue:=FALSE;
// 					ELSE
// 						GV_Axes.stAxisY.bWritebValue:=TRUE;
// 					END_IF
// 				ELSIF GV_HMI.stAxes.rtButtonMaxSofltLimit.Q THEN
// 					GV_Axes.stAxisY.mcAxisWriteParameterb:=MC_AxisParameter.AxisEnMaxSoftPosLimit;
// 					IF GV_Axes.stAxisY.bReadEnMaxSoftPosLimit THEN
// 						GV_Axes.stAxisY.bWritebValue:=FALSE;
// 					ELSE
// 						GV_Axes.stAxisY.bWritebValue:=TRUE;
// 					END_IF
// 				END_IF
// 			END_IF
		(*WriteParameter LREAL*)
// 			bAxisYWrite1:=FALSE;
// 			bAxisYWrite2:=FALSE;
// 			bAxisYWrite3:=FALSE;
// 			bAxisYWrite4:=FALSE;
// 			IF GV_Tool_Magazine.stManipulator.ePositionMag=ENUM_Position_Magazine.Top THEN
// 				IF GV_Tool_Magazine.stManipulator.lrYPosition<>GV_Tool_Magazine.stManipulator.lrYTunnel THEN
// 					GV_Axes.stAxisY.lrValueMax:=-10;
// 					GV_Axes.stAxisY.lrValueMin:=-350;
// 					bAxisYWrite1:=TRUE;
// 				ELSE
// 					GV_Axes.stAxisY.lrValueMax:=-10;
// 					GV_Axes.stAxisY.lrValueMin:=-800;
// 					bAxisYWrite2:=TRUE;
// 				END_IF
// 			END_IF
// 			IF GV_Tool_Magazine.stManipulator.ePositionMag=ENUM_Position_Magazine.Bottom THEN
// 				IF GV_Tool_Magazine.stManipulator.lrYPosition<>GV_Tool_Magazine.stManipulator.lrYTunnel THEN
// 					GV_Axes.stAxisY.lrValueMax:=-450;
// 					GV_Axes.stAxisY.lrValueMin:=-800;
// 					bAxisYWrite3:=TRUE;
// 				ELSE
// 					GV_Axes.stAxisY.lrValueMax:=-10;
// 					GV_Axes.stAxisY.lrValueMin:=-800;
// 					bAxisYWrite4:=TRUE;
// 				END_IF
// 			END_IF
// 			rtAxisYWrite1(CLK:=bAxisYWrite1);
// 			rtAxisYWrite2(CLK:=bAxisYWrite2);
// 			rtAxisYWrite3(CLK:=bAxisYWrite3);
// 			rtAxisYWrite4(CLK:=bAxisYWrite4);
// 			IF rtAxisYWrite1.Q OR rtAxisYWrite2.Q OR rtAxisYWrite3.Q OR rtAxisYWrite4.Q THEN
// 				GV_Axes.stAxisY.mcAxisWriteParameterlr:=MC_AxisParameter.AxisMaxSoftPosLimit;
// 				GV_Axes.stAxisY.lrWritelrValue:=GV_Axes.stAxisY.lrValueMax;
// 				bAxisYWriteMin:=FALSE;
// 				bAxisYWriteMax:=TRUE;
// 			END_IF
// 			IF bAxisYWriteMax AND GV_Axes.stAxisY.bWritelrBusy THEN
// 				GV_Axes.stAxisY.mcAxisWriteParameterlr:=MC_AxisParameter.AxisMinSoftPosLimit;
// 				GV_Axes.stAxisY.lrWritelrValue:=GV_Axes.stAxisY.lrValueMin;
// 				bAxisYWriteMin:=TRUE;
// 				bAxisYWriteMax:=FALSE;
// 			END_IF
// 			IF bAxisYWriteMin AND GV_Axes.stAxisY.bWritelrBusy THEN
// 				bAxisYWriteMin:=FALSE;
// 				bAxisYWriteMax:=FALSE;
// 			END_IF
// 			GV_Axes.stAxisY.bWritelrExecute:=(bAxisYWriteMax OR bAxisYWriteMin) AND GV_Axes.stAxisY.bWritelrDone AND (NOT GV_Axes.stAxisY.bWritelrBusy) AND GV_Axes.stAxisY.stDriveAx8206.AxisRef.Status.Operational;
// 			
	(* Fb *)
		IF GV_Axes.stAxisY.bPresence THEN
			fbAxisY(
					stAxis:=GV_Axes.stAxisY,
					);
		END_IF

